# B&R Automation Studio project EFI (part 21)

#### AlarmsSummary.st
```iecst
ACTION AlarmsSummary:

	gMachine.Al.xAlrDisableGoToProduction := FALSE;

	IF gMachine.Pt.CT.iNumBlocks = 1 THEN
		gMachine.Al.xAlrSafetySystemEStop:=	gBlock[1].Al.xAlrEmergencyStop;
	ELSIF gMachine.Pt.CT.iNumBlocks = 2 THEN
		gMachine.Al.xAlrSafetySystemEStop:= gBlock[1].Al.xAlrEmergencyStop OR gBlock[2].Al.xAlrEmergencyStop;
	END_IF

	iReasonSafetySystemGeneral.0 := gMachine.Al.xAlrSafetySystemEStop;
	iReasonSafetySystemGeneral.1 := gBlock[1].AlSummary.xAlrSafetySystemGeneral AND gBlock[1].parSw.xEnableToMovements;
	iReasonSafetySystemGeneral.2 := gBlock[2].AlSummary.xAlrSafetySystemGeneral AND gBlock[2].parSw.xEnableToMovements;
	iReasonSafetySystemGeneral.3 := gMachine.Al.Alarm.xAlrSafetyNotEnabled;
	gMachine.AlSummary.xAlrSafetySystemGeneral:= iReasonSafetySystemGeneral > 0;

	iReasonSafetyCutAir.0 := gBlock[1].AlSummary.xAlrSafetyCutAir AND gBlock[1].parSw.xEnableToMovements;
	iReasonSafetyCutAir.1 := gBlock[2].AlSummary.xAlrSafetyCutAir AND gBlock[2].parSw.xEnableToMovements;
	gMachine.AlSummary.xAlrSafetyCutAir:= iReasonSafetyCutAir > 0;

	//////////////////
	// General Summary
	//////////////////

	//Silvia: any general warning+any block warning+any inks warning+any photocell warning.
	//Warnings//
	reasonAnyWarningGen.0 := gMachine.Al.Warning.xNotLoadedImage;
	reasonAnyWarningGen.1 := gMachine.Al.Alarm.xAlarmPlarformInc;
	reasonAnyWarningGen.2 := gMachine.Al.Alarm.xNoActionDangerCollision;
	reasonAnyWarningGen.3 := gMachine.Al.Warning.xBentTile;
	reasonAnyWarningGen.4 := gMachine.Al.Warning.xMaxMovsBentTile;
	reasonAnyWarningGen.5 := gMachine.Al.Alarm.xAlarmNotInPrintPosition;
	reasonAnyWarningGen.6 := gMachine.Al.Warning.xExternalCleanActive;
	reasonAnyWarningGen.7 := gMachine.Al.Warning.xSAIFault;
	reasonAnyWarningGen.8 := gMachine.Al.Warning.xSAIBypass;
	reasonAnyWarningGen.9 := gMachine.Al.Warning.xSAILowBat;
	reasonAnyWarningGen.10 := gMachine.Al.Warning.xValidConfiguration;
	reasonAnyWarningGen.11 := gBelt.AlSummary.xAnyWarning;
	reasonAnyWarningGen.12 := gBlock[1].AlSummary.xAnyWarning;
	reasonAnyWarningGen.13 := gBlock[2].AlSummary.xAnyWarning;
	reasonAnyWarningGen.14 := gPhotoCells.AlSummary.xAnyWarning;
	reasonAnyWarningGen.15 := gMachine.Al.Warning.xPCCabineSensAlrm;
	reasonAnyWarningGen.16 := gCuringLed[iIndexWhiteCuringLedBar].AlSummary.xAnyWarning;
	reasonAnyWarningGen.17 := gCuringLed[iIndexColorCuringLedBar].AlSummary.xAnyWarning;
	reasonAnyWarningGen.18 := gTransVacuum[1].AlSummary.xAnyWarning;
	reasonAnyWarningGen.19 := gTransVacuum[2].AlSummary.xAnyWarning;
	reasonAnyWarningGen.20 := gMachine.parSw.UI.xWarningCondition;
	reasonAnyWarningGen.21 := gMachine.Al.Warning.xNoCleaningModeEnabled;
	reasonAnyWarningGen.22 := gMachine.Al.Warning.xMediaIncoherenceDetectedL1;
	reasonAnyWarningGen.23 := gMachine.Al.Warning.xMediaIncoherenceDetectedL2;
	reasonAnyWarningGen.24 := gMachine.Al.Warning.xAlrHoopersSoftStarterFault;
	reasonAnyWarningGen.25 := gMachine.Al.Warning.xOvervoltage;
	reasonAnyWarningGen.25 := gBeltClean.AlSummary.xAnyAlarm;
	reasonAnyWarningGen.26 := gMachine.Al.Warning.xIonAntiStatic;
	reasonAnyWarningGen.27 := gMachine.Al.Warning.xErrorAntiStatic;
	reasonAnyWarningGen.28 := gMachine.Al.Warning.xWasteInkTankMaxLevelReached;

	reasonAnyWarningInks.0 := gInks[1].AlSummary.xAnyWarning;
	reasonAnyWarningInks.1 := gInks[2].AlSummary.xAnyWarning;
	reasonAnyWarningInks.2 := gInks[3].AlSummary.xAnyWarning;
	reasonAnyWarningInks.3 := gInks[4].AlSummary.xAnyWarning;
	reasonAnyWarningInks.4 := gInks[5].AlSummary.xAnyWarning;
	reasonAnyWarningInks.5 := gInks[6].AlSummary.xAnyWarning;
	reasonAnyWarningInks.6 := gInks[7].AlSummary.xAnyWarning;
	reasonAnyWarningInks.7 := gInks[8].AlSummary.xAnyWarning;
	reasonAnyWarningInks.8 := gInks[9].AlSummary.xAnyWarning;
	reasonAnyWarningInks.9 := gInks[10].AlSummary.xAnyWarning;
	reasonAnyWarningInks.10 := gInks[11].AlSummary.xAnyWarning;
	reasonAnyWarningInks.11 := gInks[12].AlSummary.xAnyWarning;

	gMachine.AlSummary.xAnyWarning:= reasonAnyWarningGen>0 OR reasonAnyWarningInks>0;

	//Any ALarm//
	gMachine.AlSummary.xAnyAlarm:= 	gMachine.AlSummary.xAlarmCritical OR
									gMachine.AlSummary.xAlarmStop;

	//Critial alarms//
	iReasonCritical.0 := gMachine.AlSummary.xAlrSafetySystemGeneral;
	iReasonCritical.1 := gMachine.Al.Alarm.xAlarmSAIPowerOff;
	iReasonCritical.2 := gBelt.AlSummary.xAlarmCritical;
	iReasonCritical.3 := gBlock[1].AlSummary.xAlarmCritical;
	iReasonCritical.4 := gBlock[2].AlSummary.xAlarmCritical;
	iReasonCritical.5 := gMachine.Al.Alarm.xAlrWrongPhysConf;
	iReasonCritical.6 := gMachine.Al.Alarm.xNoPowered;

	gMachine.AlSummary.CurrentReasonCritical := iReasonCritical;

	gMachine.AlSummary.xAlarmCritical:=  iReasonCritical > 0;
	//Register the reason of the Critical Alarm
	IF gMachine.St.Mode.xAuto AND EDGEPOS(gMachine.AlSummary.xAlarmCritical) THEN
		gMachine.AlSummary.iReasonCritical := iReasonCritical;
		LogCriticalAlarm;
	ELSIF EDGEPOS(gMachine.St.Mode.xAuto AND NOT gMachine.AlSummary.xAlarmCritical) THEN
		gMachine.AlSummary.iReasonCritical := 0;
	END_IF

	//Alarms stop//
	//Inks
	iReasonStopInks.0 := gInks[1].AlSummary.xAlarmStop;
	iReasonStopInks.1 := gInks[2].AlSummary.xAlarmStop;
	iReasonStopInks.2 := gInks[3].AlSummary.xAlarmStop;
	iReasonStopInks.3 := gInks[4].AlSummary.xAlarmStop;
	iReasonStopInks.4 := gInks[5].AlSummary.xAlarmStop;
	iReasonStopInks.5 := gInks[6].AlSummary.xAlarmStop;
	iReasonStopInks.6 := gInks[7].AlSummary.xAlarmStop;
	iReasonStopInks.7 := gInks[8].AlSummary.xAlarmStop;
	iReasonStopInks.8 := gInks[9].AlSummary.xAlarmStop;
	iReasonStopInks.9 := gInks[10].AlSummary.xAlarmStop;
	iReasonStopInks.10 := gInks[11].AlSummary.xAlarmStop;
	iReasonStopInks.11 := gInks[12].AlSummary.xAlarmStop;

	//General 1
	iReasonStopGen.0 := gMachine.Al.Alarm.xAlarmAir1;
	iReasonStopGen.1 := gMachine.Al.Alarm.xAlarmComPcPLC;
	iReasonStopGen.2 := gMachine.Al.Alarm.xAlarmEnableWithoutBarsOn;
	iReasonStopGen.3 := gMachine.Al.Alarm.xAlarmMountedPiece;
	iReasonStopGen.4 := gMachine.Al.Alarm.xAlarmSAIPowerFault;
	iReasonStopGen.5 := gMachine.Al.xAlrSafetySystemEStop;
	iReasonStopGen.6 := gMachine.Al.Alarm.xAlrThicknSystemNotSelected;
	iReasonStopGen.7 := gBlock[1].AlSummary.xAlarmStop;
	iReasonStopGen.8 := gBlock[2].AlSummary.xAlarmStop;
	iReasonStopGen.9 := gBelt.AlSummary.xAlarmStop;
	iReasonStopGen.10 := gDing.AlSummary.xAlarmStop;
	iReasonStopGen.11 := gPhotoCells.AlSummary.xAlarmStop;
	iReasonStopGen.12 := gTransVacuum[1].AlSummary.xAlarmStop;
	iReasonStopGen.13 := gTransVacuum[2].AlSummary.xAlarmStop;
	iReasonStopGen.14 := gMachine.Al.Alarm.xPDBrokenSensorL1;
	iReasonStopGen.15 := gMachine.Al.Alarm.xPDBrokenSensorL2;
	iReasonStopGen.16 := gJamDetect[1].AlSummary.xAlarmStop;
	iReasonStopGen.17 := gJamDetect[2].AlSummary.xAlarmStop;
	iReasonStopGen.18 := gNonCrash[1].AlSummary.xAlarmStop;
	iReasonStopGen.19 := gNonCrash[2].AlSummary.xAlarmStop;
	iReasonStopGen.20 := gMachine.Al.Alarm.xAlr24Vdc;
	//When printer is controlled by line, we consider curing led lamps errors in LineCtrl to execute a ControlledStop, but when printer is running by its own, must stop inmediately
	iReasonStopGen.21 := (gCuringLed[iIndexWhiteCuringLedBar].AlSummary.xAlarmStop OR gCuringLed[iIndexWhiteCuringLedBar].AlSummary.xAlarmCritical) AND NOT gMachine.Pt.xControlledByLine;
	iReasonStopGen.22 := (gCuringLed[iIndexColorCuringLedBar].AlSummary.xAlarmStop OR gCuringLed[iIndexColorCuringLedBar].AlSummary.xAlarmCritical) AND NOT gMachine.Pt.xControlledByLine;
	iReasonStopGen.23 := gMachine.Al.Alarm.xAlrDingWrongPosition;
	iReasonStopGen.24 := gMachine.Al.Alarm.xSwCriticalCondition;
	iReasonStopGen.25 := gJamDetect[3].AlSummary.xAlarmStop;
	iReasonStopGen.26 := gMachine.Al.Alarm.xNotLoadedImage;
	iReasonStopGen.27 := gThicknessCtrl.AlSummary.xAlarmStop;
	iReasonStopGen.28 := gMachine.Al.Alarm.xAlrThickOutLimits;
	iReasonStopGen.29 := gMachine.Al.Alarm.xAlrLengthOutLimits;
	iReasonStopGen.30 := gMachine.Al.Alarm.xAlrWidthOutLimits;

	gMachine.AlSummary.CurrentReasonStop[0] := iReasonStopInks;
	gMachine.AlSummary.CurrentReasonStop[1] := iReasonStopGen;

	gMachine.AlSummary.xAlarmStop:= iReasonStopGen > 0 OR iReasonStopInks > 0;
	//Register the reason of the Alarm
	IF NOT gMachine.St.AutoMode.xStop AND EDGEPOS(gMachine.AlSummary.xAlarmStop) THEN
		gMachine.AlSummary.iReasonStop[0] := iReasonStopInks;
		gMachine.AlSummary.iReasonStop[1] := iReasonStopGen;
		LogStopAlarm;
	ELSIF EDGEPOS(NOT gMachine.St.AutoMode.xStop AND NOT gMachine.AlSummary.xAlarmStop) THEN
		gMachine.AlSummary.iReasonStop[0] := 0;
		gMachine.AlSummary.iReasonStop[1] := 0;
	END_IF

END_ACTION
```

#### MachineInputs.st
```iecst
ACTION MachineInputs:

	// Product Detect. Manage general signal from signal connected to any block

	//Aggregated signals in the machine to clarify reading code
	CASE gMachine.Pt.PDSignalTpe OF
		PDCFG_CARRIAGE:
			// Check proper data assigned
			IF gMachine.In.ProductDetect.pPDCarriageSignalL1 = 0 OR gMachine.In.ProductDetect.pPDCarriageSignalL2 = 0 THEN
				RETURN;
			END_IF
			// Data pointer assignation
			xPDCarriageL1 ACCESS gMachine.In.ProductDetect.pPDCarriageSignalL1;
			xPDCarriageL2 ACCESS gMachine.In.ProductDetect.pPDCarriageSignalL2;
			// Status assignation
			gMachine.St.ProductDetect.xProductDetectL1 := xPDCarriageL1;
			gMachine.St.ProductDetect.xProductDetectL2 := xPDCarriageL2;

		PDCFG_SENSOR_AND_CARRIAGE,
		PDCFG_SENSOR:
			// Check proper data assigned
			IF gMachine.In.ProductDetect.pPDSignalSensorL1 = 0 OR ((gMachine.In.ProductDetect.pPDSignalSensorL2 = 0) AND gMachine.Pt.Hw.xDoubleLineAllowed) THEN
				RETURN;
			END_IF

			// Data pointer assignation
			xPDSignalSensorL1 ACCESS gMachine.In.ProductDetect.pPDSignalSensorL1;
			IF gMachine.Pt.Hw.xDoubleLineAllowed THEN
				xPDSignalSensorL2 ACCESS gMachine.In.ProductDetect.pPDSignalSensorL2;
			END_IF

			IF gThicknessCtrl.parameters.Detection.ProductDetect.xLoadMedia THEN
				gMachine.St.ProductDetect.xProductDetectL1 := gThicknessCtrl.status.Detection.xFilteredProductDetectMediaL1 AND gMachine.St.Position.xInPrint AND gMachine.parSw.Electronics.xRobotReadyL1;
				gMachine.St.ProductDetect.xProductDetectL2 := gThicknessCtrl.status.Detection.xFilteredProductDetectMediaL2 AND gMachine.St.Position.xInPrint AND gMachine.parSw.Electronics.xRobotReadyL2;
			ELSE
				//Status assignation
				gMachine.St.ProductDetect.xProductDetectL1 := xPDSignalSensorL1 AND gMachine.St.Position.xInPrint AND gMachine.parSw.Electronics.xRobotReadyL1;
				gMachine.St.ProductDetect.xProductDetectL2 := xPDSignalSensorL2 AND gMachine.St.Position.xInPrint AND gMachine.parSw.Electronics.xRobotReadyL2;
			END_IF

	END_CASE

	gMachine.St.ProductDetect.xAnyProductDetect := gMachine.St.ProductDetect.xProductDetectL1 OR gMachine.St.ProductDetect.xProductDetectL2;
	gMachine.St.ProductDetect.xAnyProductDetectDtpStricted := gMachine.St.ProductDetect.xProductDetectL1 OR (gMachine.St.ProductDetect.xProductDetectL2 AND gMachine.parSw.Dtp.xDoubleLine);

	gMachine.St.xMediaDetected := gDing.In.xDingLow OR gPhotoCells.status.xLowPieceDetect;

	//Counting edges of Product Detect sensor
	IF EDGEPOS(gMachine.St.ProductDetect.xProductDetectL1) THEN
		diCountProductDetectEdgesL1 := diCountProductDetectEdgesL1 + 1;
	END_IF
	IF EDGEPOS(gMachine.St.ProductDetect.xProductDetectL2) THEN
		diCountProductDetectEdgesL2 := diCountProductDetectEdgesL2 + 1;
	END_IF

	//Just for testing. To simulate media in real machine while degbugging with no real media available
	IF (gSimMachine.Commands.Media.xContinuousMediaPresent AND gBelt.states.xRuningBelt) THEN
		xBeltSpeedChanged 	:= rPrevBeltSpeed <> gBelt.states.rCurrentSpeed;
		xFormatChanged 		:= 	rPrevBoardLength <> gMachine.parSw.Media.rLength OR
								rPrevBoardGap <> gMachine.parSw.Media.rGap;

		IF (xBeltSpeedChanged OR xFormatChanged) AND (gBelt.states.rCurrentSpeed > gc_rMinSpeedToStart) THEN
			rBeltSpeedMmMs := (gBelt.states.rCurrentSpeed/60);

			//Board
			tiBoardTime := REAL_TO_TIME(gMachine.parSw.Media.rLength/rBeltSpeedMmMs);
			tiGapTime := REAL_TO_TIME(gMachine.parSw.Media.rGap/rBeltSpeedMmMs);

		END_IF
		rPrevBeltSpeed := gBelt.states.rCurrentSpeed;
		rPrevBoardLength := gMachine.parSw.Media.rLength;
		rPrevBoardGap := gMachine.parSw.Media.rGap;
		rPrevStainLength := gSimMachine.Parameters.rStainLength;
		rPrevStainGap := gSimMachine.Parameters.rStainGap;

		//To simulate a media
		BoardsFeedMinGap.tTimeOn := tiBoardTime;
		BoardsFeedMinGap.tTimeOff := tiGapTime;
		BoardsFeedMinGap.xEnable := TRUE;
	ELSE
		BoardsFeedMinGap.xEnable := FALSE;
	END_IF
	BoardsFeedMinGap();
END_ACTION
```

#### ResetAlarms.st
```iecst
ACTION ResetAlarms:

	gMachine.Al:=stPrinterAlarmsReseted;
	gMachine.Al.Alarm:= stPrinterAlarmsListReseted;

END_ACTION
```

- MachineStates.graphml - YED documentation (not shown)

### Program Logical/Printer/PhysicalMapping/PhysicalMapInputs (IEC) - Inputs program

#### Variables.var
```iecst
VAR
	T_Mute : TOF;
	T_Reset : TON;
	iIndexBlock : USINT;
	iIndexVac : USINT;
	iIndexCuringLed : USINT;
END_VAR
```

#### InputsNozomi2.st
```iecst
ACTION InputsNozomi2:

	//////////
	//PRINTER
	//////////

	// Machine controlled by line. Always with consent
	gMachine.In.xConsentL1Ok := TRUE;
	gMachine.In.xConsentL2Ok := TRUE;

	//Digital Inputs
	gMachine.In.Buttons.xStart := X20DIF371_101.DInput[1];
	gMachine.In.Buttons.xStop := NOT X20DIF371_101.DInput[2];
	gMachine.In.Buttons.xAuto := X20DIF371_101.DInput[3];
	gMachine.In.Buttons.xZero := NOT X20DIF371_101.DInput[4];
	gMachine.In.Buttons.xManual := X20DIF371_101.DInput[5];
	gMachine.In.Buttons.xReset := X20DIF371_101.DInput[6];

	gMachine.In.ProductDetect.pPDCarriageSignalL1 := ADR(X20DIF371_101.DInput[7]);
	gMachine.In.ProductDetect.pPDCarriageSignalL2 := ADR(X20DIF371_101.DInput[8]);
	gMachine.In.ProductDetect.pPDCarriage2SignalL1 := ADR(X20DIF371_101.DInput[9]);
	gMachine.In.ProductDetect.pPDCarriage2SignalL2 := ADR(X20DIF371_101.DInput[10]);

	//Jam device N3
	gJamInputs[3].xJamLowCrash := X20DIF371_101.DInput[11];
	gJamInputs[3].xJamTestOk := X20DIF371_101.DInput[12];
	gJamInputs[3].xJamCrash[1] := X20DIF371_101.DInput[13];

	gInksInputs[1].xPrintHeadsPsuOK := X20DIF371_102.DInput[1];
	gInksInputs[2].xPrintHeadsPsuOK := X20DIF371_102.DInput[2];
	gInksInputs[3].xPrintHeadsPsuOK := X20DIF371_102.DInput[3];
	gInksInputs[4].xPrintHeadsPsuOK := X20DIF371_102.DInput[4];
	gInksInputs[5].xPrintHeadsPsuOK := X20DIF371_102.DInput[5];
	gInksInputs[6].xPrintHeadsPsuOK := X20DIF371_102.DInput[6];
	gInksInputs[7].xPrintHeadsPsuOK := X20DIF371_102.DInput[7];
	gInksInputs[8].xPrintHeadsPsuOK := X20DIF371_102.DInput[8];
	//SPARE := NOT X20DIF371_102.DInput[9];
	gBelt.parameters.xDriveProtectionOK := X20DIF371_102.DInput[10];
	gBlockInputs[1].xDriveProtectionOK := gBlockInputs[1].xDifferentialOK := X20DIF371_102.DInput[11];
	//Non-crash - CB contact alarm := X20DIF371_102.DInput[12];
	gMachine.In.x24Vdc := X20DIF371_102.DInput[13];
	gBlockInputs[1].xReferenceDI := X20DIF371_102.DInput[14];
	//Back Safety Key unlock - PRINTER := X20DIF371_102.DInput[15];
	gMachine.In.xCameraDefectDetected := X20DIF371_102.DInput[16];

	IF NOT gMachine.St.HwData.xUpsOutOfPrinter THEN
		gMachine.In.UPSs[1].LoadOnUtility	:= X20DIF371_103.DInput[1];
		gMachine.In.UPSs[1].LoadOnBattery 	:= gMachine.In.UPSs[1].xPowerFault := X20DIF371_103.DInput[2]; //To review why name of signal is different for S1400 than Nz2. Signal coming from ups has same behaviour
		gMachine.In.UPSs[1].xLowBattery 	:= X20DIF371_103.DInput[3];
		gMachine.In.UPSs[1].xByPass 		:= X20DIF371_103.DInput[4];
		gMachine.In.UPSs[2].LoadOnUtility	:= X20DIF371_103.DInput[5];
		gMachine.In.UPSs[2].LoadOnBattery 	:= gMachine.In.UPSs[2].xPowerFault := X20DIF371_103.DInput[6]; //To review why name of signal is different for S1400 than Nz2. Signal coming from ups has same behaviour
		gMachine.In.UPSs[2].xLowBattery 	:= X20DIF371_103.DInput[7];
		gMachine.In.UPSs[2].xByPass 		:= X20DIF371_103.DInput[8];
	END_IF

	gMachine.In.ProductDetect.pPDSignalSensorL1	:= ADR(X20DIF371_103.DInput[9]);
	gMachine.In.ProductDetect.pPDSignalSensorL2	:= ADR(X20DIF371_103.DInput[10]);
//	gPhotoCells.Inputs.Signals.xPhotoCells[1] := NOT X20DIF371_103.DInput[11]; //Signal moved to FastInputs program
//	gPhotoCells.Inputs.Signals.xPhotoCells[2] := NOT X20DIF371_103.DInput[12]; //Signal moved to FastInputs program
//	gPhotoCells.Inputs.Signals.xPhotoCells[3] := NOT X20DIF371_103.DInput[13]; //Signal moved to FastInputs program
//	gPhotoCells.Inputs.Signals.xPhotoCells[4] := NOT X20DIF371_103.DInput[14]; //Signal moved to FastInputs program
//	gPhotoCells.Inputs.Signals.xPhotoCells[5] := NOT X20DIF371_103.DInput[15]; //Signal moved to FastInputs program
//	gPhotoCells.Inputs.Signals.xPhotoCells[6] := NOT X20DIF371_103.DInput[16]; //Signal moved to FastInputs program

	gInksInputs[1].xKlixonTriggered := X20DIF371_104.DInput[1];
	gInksInputs[2].xKlixonTriggered := X20DIF371_104.DInput[2];
	gInksInputs[3].xKlixonTriggered := X20DIF371_104.DInput[3];
	gInksInputs[4].xKlixonTriggered := X20DIF371_104.DInput[4];
	gInksInputs[5].xKlixonTriggered := X20DIF371_104.DInput[5];
	gInksInputs[6].xKlixonTriggered := X20DIF371_104.DInput[6];
	gInksInputs[7].xKlixonTriggered := X20DIF371_104.DInput[7];
	gInksInputs[8].xKlixonTriggered := X20DIF371_104.DInput[8];
	gJamInputs[1].xJamCrash[1] := X20DIF371_104.DInput[9];
	gJamInputs[1].xJamCrash[2] := X20DIF371_104.DInput[10];
	gJamInputs[1].xJamCrash[3] := X20DIF371_104.DInput[11];
	gJamInputs[1].xJamCrash[4] := X20DIF371_104.DInput[12];
	gJamInputs[2].xJamCrash[1] := X20DIF371_104.DInput[13];
	gJamInputs[2].xJamCrash[2] := X20DIF371_104.DInput[14];
	gJamInputs[2].xJamCrash[3] := X20DIF371_104.DInput[15];
	gJamInputs[2].xJamCrash[4] := X20DIF371_104.DInput[16];

	gInksInputs[1].xOverpressure  := NOT X20DIF371_105.DInput[1];
	gInksInputs[2].xOverpressure  := NOT X20DIF371_105.DInput[2];
	gInksInputs[3].xOverpressure  := NOT X20DIF371_105.DInput[3];
	gInksInputs[4].xOverpressure  := NOT X20DIF371_105.DInput[4];
	gInksInputs[5].xOverpressure  := NOT X20DIF371_105.DInput[5];
	gInksInputs[6].xOverpressure  := NOT X20DIF371_105.DInput[6];
	gInksInputs[7].xOverpressure  := NOT X20DIF371_105.DInput[7];
	gInksInputs[8].xOverpressure  := NOT X20DIF371_105.DInput[8];
	//Spare := X20DIF371_105.DInput[9];
	//Spare := X20DIF371_105.DInput[10];
	gMachine.In.xDegasserPressure := X20DIF371_105.DInput[11];
	gJamInputs[1].xJamLowCrash := X20DIF371_105.DInput[12];
	gJamInputs[2].xJamLowCrash := X20DIF371_105.DInput[13];
	gJamInputs[1].xJamTestOk := X20DIF371_105.DInput[14];
	gJamInputs[2].xJamTestOk := X20DIF371_105.DInput[15];
	FOR iIndexCuringLed:=1 TO MAX_LAST_CURING_LED DO
		gCuringLed[iIndexCuringLed].Signals.Inputs.xFrontDoorClosed := X20DIF371_105.DInput[16];
	END_FOR
	gBlockInputs[1].xFrontDoorClosed := X20DIF371_105.DInput[16];

	gBlockInputs[1].xPrintHeadPSU[1] := X20DI9372_107.DInput[1];
	gBlockInputs[1].xPrintHeadPSU[2] := X20DI9372_107.DInput[2];
	gBlockInputs[1].xPrintHeadPSU[3] := X20DI9372_107.DInput[3];
	gBlockInputs[1].xPrintHeadPSU[4] := X20DI9372_107.DInput[4];
	gBlockInputs[1].xPrintHeadPSU[5] := X20DI9372_107.DInput[5];
	gBlockInputs[1].xPrintHeadPSU[6] := X20DI9372_107.DInput[6];
	gBlockInputs[1].xHeaterDcOkBusBar1 := X20DI9372_107.DInput[7];
	gBlockInputs[1].xHeaterDcOkBusBar2 := X20DI9372_107.DInput[8];
	gMachine.In.xWasteInkTankMaxLevelReached := X20DI9372_107.DInput[9];

	//Analog inputs
	gInksInputs[1].iVacuum1Raw := X20AI8321_111.AInput[1];
	gInksInputs[1].xVacuum1SensorError 	:= StatusAnalogInputBroken( X20AI8321_111.ModuleOk, X20AI8321_111.Status01, X20AI8321_111.Status02, 1);
	gInksInputs[1].iVacuum2Raw := X20AI8321_111.AInput[2];
	gInksInputs[1].xVacuum2SensorError 	:= StatusAnalogInputBroken( X20AI8321_111.ModuleOk, X20AI8321_111.Status01, X20AI8321_111.Status02, 2);
	gInksInputs[2].iVacuum1Raw := X20AI8321_111.AInput[3];
	gInksInputs[2].xVacuum1SensorError 	:= StatusAnalogInputBroken( X20AI8321_111.ModuleOk, X20AI8321_111.Status01, X20AI8321_111.Status02, 3);
	gInksInputs[2].iVacuum2Raw := X20AI8321_111.AInput[4];
	gInksInputs[2].xVacuum2SensorError 	:= StatusAnalogInputBroken( X20AI8321_111.ModuleOk, X20AI8321_111.Status01, X20AI8321_111.Status02, 4);
	gInksInputs[3].iVacuum1Raw := X20AI8321_111.AInput[5];
	gInksInputs[3].xVacuum1SensorError 	:= StatusAnalogInputBroken( X20AI8321_111.ModuleOk, X20AI8321_111.Status01, X20AI8321_111.Status02, 5);
	gInksInputs[3].iVacuum2Raw := X20AI8321_111.AInput[6];
	gInksInputs[3].xVacuum2SensorError 	:= StatusAnalogInputBroken( X20AI8321_111.ModuleOk, X20AI8321_111.Status01, X20AI8321_111.Status02, 6);
	gInksInputs[4].iVacuum1Raw := X20AI8321_111.AInput[7];
	gInksInputs[4].xVacuum1SensorError 	:= StatusAnalogInputBroken( X20AI8321_111.ModuleOk, X20AI8321_111.Status01, X20AI8321_111.Status02, 7);
	gInksInputs[4].iVacuum2Raw := X20AI8321_111.AInput[8];
	gInksInputs[4].xVacuum2SensorError 	:= StatusAnalogInputBroken( X20AI8321_111.ModuleOk, X20AI8321_111.Status01, X20AI8321_111.Status02, 8);

	gInksInputs[5].iVacuum1Raw := X20AI8321_112.AInput[1];
	gInksInputs[5].xVacuum1SensorError 	:= StatusAnalogInputBroken( X20AI8321_112.ModuleOk, X20AI8321_112.Status01, X20AI8321_112.Status02, 1);
	gInksInputs[5].iVacuum2Raw := X20AI8321_112.AInput[2];
	gInksInputs[5].xVacuum2SensorError 	:= StatusAnalogInputBroken( X20AI8321_112.ModuleOk, X20AI8321_112.Status01, X20AI8321_112.Status02, 2);
	gInksInputs[6].iVacuum1Raw := X20AI8321_112.AInput[3];
	gInksInputs[6].xVacuum1SensorError 	:= StatusAnalogInputBroken( X20AI8321_112.ModuleOk, X20AI8321_112.Status01, X20AI8321_112.Status02, 3);
	gInksInputs[6].iVacuum2Raw := X20AI8321_112.AInput[4];
	gInksInputs[6].xVacuum2SensorError 	:= StatusAnalogInputBroken( X20AI8321_112.ModuleOk, X20AI8321_112.Status01, X20AI8321_112.Status02, 4);
	gInksInputs[7].iVacuum1Raw := X20AI8321_112.AInput[5];
	gInksInputs[7].xVacuum1SensorError 	:= StatusAnalogInputBroken( X20AI8321_112.ModuleOk, X20AI8321_112.Status01, X20AI8321_112.Status02, 5);
	gInksInputs[7].iVacuum2Raw := X20AI8321_112.AInput[6];
	gInksInputs[7].xVacuum2SensorError 	:= StatusAnalogInputBroken( X20AI8321_112.ModuleOk, X20AI8321_112.Status01, X20AI8321_112.Status02, 6);
	gInksInputs[8].iVacuum1Raw := X20AI8321_112.AInput[7];
	gInksInputs[8].xVacuum1SensorError 	:= StatusAnalogInputBroken( X20AI8321_112.ModuleOk, X20AI8321_112.Status01, X20AI8321_112.Status02, 7);
	gInksInputs[8].iVacuum2Raw := X20AI8321_112.AInput[8];
	gInksInputs[8].xVacuum2SensorError 	:= StatusAnalogInputBroken( X20AI8321_112.ModuleOk, X20AI8321_112.Status01, X20AI8321_112.Status02, 8);

	gTransVacuum[1].Inputs.iPressureRaw := X20AI8321_113.AInput[1];
	gTransVacuum[1].Inputs.xPressureSensorError := StatusAnalogInputBroken( X20AI8321_113.ModuleOk, X20AI8321_113.Status01, X20AI8321_113.Status02, 1);
	gTransVacuum[2].Inputs.iPressureRaw := X20AI8321_113.AInput[2];
	gTransVacuum[2].Inputs.xPressureSensorError := StatusAnalogInputBroken( X20AI8321_113.ModuleOk, X20AI8321_113.Status01, X20AI8321_113.Status02, 2);

	gInksInputs[2].iInTankLevel := X20AI8321_113.AInput[3];
	gInksInputs[2].xInkLevelTankSensorError := StatusAnalogInputBroken( X20AI8321_113.ModuleOk, X20AI8321_113.Status01, X20AI8321_113.Status02, 3);
	gInksInputs[3].iInTankLevel := X20AI8321_113.AInput[4];
	gInksInputs[3].xInkLevelTankSensorError := StatusAnalogInputBroken( X20AI8321_113.ModuleOk, X20AI8321_113.Status01, X20AI8321_113.Status02, 4);
	gInksInputs[4].iInTankLevel := X20AI8321_113.AInput[5];
	gInksInputs[4].xInkLevelTankSensorError := StatusAnalogInputBroken( X20AI8321_113.ModuleOk, X20AI8321_113.Status01, X20AI8321_113.Status02, 5);
	gInksInputs[5].iInTankLevel := X20AI8321_113.AInput[6];
	gInksInputs[5].xInkLevelTankSensorError := StatusAnalogInputBroken( X20AI8321_113.ModuleOk, X20AI8321_113.Status01, X20AI8321_113.Status02, 6);
	gInksInputs[6].iInTankLevel := X20AI8321_113.AInput[7];
	gInksInputs[6].xInkLevelTankSensorError := StatusAnalogInputBroken( X20AI8321_113.ModuleOk, X20AI8321_113.Status01, X20AI8321_113.Status02, 7);
	IF (gMachine.Pt.MachineModel = Type_NOZ_2_AQ) THEN
		gInksInputs[7].iInTankLevel := X20AI8321_113.AInput[8];
		gInksInputs[7].xInkLevelTankSensorError := StatusAnalogInputBroken( X20AI8321_113.ModuleOk, X20AI8321_113.Status01, X20AI8321_113.Status02, 8);
	ELSE
		gInksInputs[8].iInTankLevel := X20AI8321_113.AInput[8];
		gInksInputs[8].xInkLevelTankSensorError := StatusAnalogInputBroken( X20AI8321_113.ModuleOk, X20AI8321_113.Status01, X20AI8321_113.Status02, 8);
	END_IF

	//PT100
	gBlockInputs[1].xModuleTemp01Ok	:= X20AT4222_118.ModuleOk;
	gInksInputs[1].iTemperatureRaw := X20AT4222_118.TempInput[1];
	gInksInputs[1].xTempSensorError	:= StatusTemperatureInput(X20AT4222_118.Status01, 1);
	gInksInputs[2].iTemperatureRaw := X20AT4222_118.TempInput[2];
	gInksInputs[2].xTempSensorError	:= StatusTemperatureInput(X20AT4222_118.Status01, 2);
	gInksInputs[3].iTemperatureRaw := X20AT4222_118.TempInput[3];
	gInksInputs[3].xTempSensorError	:= StatusTemperatureInput(X20AT4222_118.Status01, 3);
	gInksInputs[4].iTemperatureRaw := X20AT4222_118.TempInput[4];
	gInksInputs[4].xTempSensorError	:= StatusTemperatureInput(X20AT4222_118.Status01, 4);

	gBlockInputs[1].xModuleTemp02Ok	:= X20AT4222_119.ModuleOk;
	gInksInputs[5].iTemperatureRaw := X20AT4222_119.TempInput[1];
	gInksInputs[5].xTempSensorError	:= StatusTemperatureInput(X20AT4222_119.Status01, 1);
	gInksInputs[6].iTemperatureRaw := X20AT4222_119.TempInput[2];
	gInksInputs[6].xTempSensorError	:= StatusTemperatureInput(X20AT4222_119.Status01, 2);
	gInksInputs[7].iTemperatureRaw := X20AT4222_119.TempInput[3];
	gInksInputs[7].xTempSensorError	:= StatusTemperatureInput(X20AT4222_119.Status01, 3);
	gInksInputs[8].iTemperatureRaw := X20AT4222_119.TempInput[4];
	gInksInputs[8].xTempSensorError	:= StatusTemperatureInput(X20AT4222_119.Status01, 4);

	// SI UNIT BK1
	gBlockInputs[1].xSiUnitModuleOk		:= SiUnitPwrLnkBK1.ModuleOk;
	gMachine.In.xAirSupply				:= SiUnitPwrLnkBK1.Input01_16.0;
	gBlockInputs[1].xAirVenturiOK		:= SiUnitPwrLnkBK1.Input01_16.1;
	gBlockInputs[1].xTrayOut			:= SiUnitPwrLnkBK1.Input01_16.2;
	gBlockInputs[1].xIclaSensor			:= SiUnitPwrLnkBK1.Input01_16.3;
	gTransVacuum[1].Inputs.xVaccAirFlow	:= gTransVacuum[2].Inputs.xVaccAirFlow := SiUnitPwrLnkBK1.Input01_16.4;
	gTransVacuum[1].Inputs.xJointSystemPressure:= gTransVacuum[2].Inputs.xJointSystemPressure := SiUnitPwrLnkBK1.Input01_16.5;
	gMachine.In.CleanBelt.xLowPosition 	:= SiUnitPwrLnkBK1.Input01_16.6;
	gMachine.In.CleanBelt.xHighPosition := SiUnitPwrLnkBK1.Input01_16.7;
	gBlockInputs[1].xBarsIn := TRUE;
	gTransVacuum[1].Inputs.xSafetyEnable := gTransVacuum[2].Inputs.xSafetyEnable := gMachine.In.xSafetyEnabled;

	//Signals Forced by Configuration
	gBlockInputs[1].Safety.xFrontEStopOK := gSafetyController.Inputs.xPrinterFrontsideEstop;
	gBlockInputs[1].Safety.xRearEStopOK := gSafetyController.Inputs.xPrinterBacksideEstop;

	gBlockInputs[1].Safety.xFrontSafetyOK	:= gSafetyController.Inputs.xPrinterFrontsideEstop AND gSafetyController.Inputs.xPrinterLightCurtain;
	gBlockInputs[1].Safety.xRearSafetyOK	:= gSafetyController.Inputs.xPrinterBacksideEstop AND gSafetyController.Inputs.xPrinterDoorLock;
	gBlockInputs[1].Safety.xSafetyOK 		:= gMachine.In.xSafetyEnabled;

	//There are no specific enables for light curtains. So we mapp PrinterLightCurtain status to these inputs to acknowledge that curtain is crossed
	gBlockInputs[1].Safety.xCurtainEnable01 := gBlockInputs[1].Safety.xCurtainEnable02 := gSafetyController.Inputs.xPrinterLightCurtain;

	//Signals Forced by Configuration
	FOR iIndexVac := 1 TO MAX_LAST_TRANS_VACUUM DO gTransVacuum[iIndexVac].Inputs.xBlowersAnyCB := FALSE; END_FOR

	///////////////////////////
	//UV Curing leds related

	//Digital inputs
	gCuringLed[iIndexColorCuringLedBar].Lamp[1].Inputs.ThermalFault	:= NOT X20DIF371_153.DInput[1];
	gCuringLed[iIndexColorCuringLedBar].Lamp[1].Inputs.SLMFault		:= NOT X20DIF371_153.DInput[2];
	gCuringLed[iIndexColorCuringLedBar].Lamp[2].Inputs.ThermalFault	:= NOT X20DIF371_153.DInput[3];
	gCuringLed[iIndexColorCuringLedBar].Lamp[2].Inputs.SLMFault		:= NOT X20DIF371_153.DInput[4];
	gCuringLed[iIndexColorCuringLedBar].Lamp[3].Inputs.ThermalFault	:= NOT X20DIF371_153.DInput[5];
	gCuringLed[iIndexColorCuringLedBar].Lamp[3].Inputs.SLMFault		:= NOT X20DIF371_153.DInput[6];
	gCuringLed[iIndexColorCuringLedBar].Lamp[4].Inputs.ThermalFault	:= NOT X20DIF371_153.DInput[7];
	gCuringLed[iIndexColorCuringLedBar].Lamp[4].Inputs.SLMFault		:= NOT X20DIF371_153.DInput[8];
	gCuringLed[iIndexColorCuringLedBar].Signals.Inputs.xN2HighFlow	:= NOT X20DIF371_153.DInput[9];
	gCuringLed[iIndexColorCuringLedBar].Signals.Inputs.xN2LowFlow		:= NOT X20DIF371_153.DInput[10];
	gMachine.In.AntiStatic.xGenAlarm								:= X20DIF371_153.DInput[13];
	gMachine.In.AntiStatic.xIonLevelAlarm							:= X20DIF371_153.DInput[14];

	gCuringLed[iIndexWhiteCuringLedBar].Lamp[1].Inputs.ThermalFault	:= NOT X20DIF371_154.DInput[1];
	gCuringLed[iIndexWhiteCuringLedBar].Lamp[1].Inputs.SLMFault		:= NOT X20DIF371_154.DInput[2];
	gCuringLed[iIndexWhiteCuringLedBar].Lamp[2].Inputs.ThermalFault	:= NOT X20DIF371_154.DInput[3];
	gCuringLed[iIndexWhiteCuringLedBar].Lamp[2].Inputs.SLMFault		:= NOT X20DIF371_154.DInput[4];
	gCuringLed[iIndexWhiteCuringLedBar].Lamp[3].Inputs.ThermalFault	:= NOT X20DIF371_154.DInput[5];
	gCuringLed[iIndexWhiteCuringLedBar].Lamp[3].Inputs.SLMFault		:= NOT X20DIF371_154.DInput[6];
	gCuringLed[iIndexWhiteCuringLedBar].Lamp[4].Inputs.ThermalFault	:= NOT X20DIF371_154.DInput[7];
	gCuringLed[iIndexWhiteCuringLedBar].Lamp[4].Inputs.SLMFault		:= NOT X20DIF371_154.DInput[8];
	gCuringLed[iIndexWhiteCuringLedBar].Signals.Inputs.xN2HighFlow	:= NOT X20DIF371_154.DInput[9];
	gCuringLed[iIndexWhiteCuringLedBar].Signals.Inputs.xN2LowFlow		:= NOT X20DIF371_154.DInput[10];

	gMachine.In.CleanBelt.xError := X20DIF371_154.DInput[13];

	gMachine.In.CleanBelt.xOpenGuide := X20DIF371_154.DInput[15]; //Clean Belt - Open Guide

	//Analog inputs
	gCuringLed[iIndexColorCuringLedBar].Lamp[1].Inputs.TemperatureRaw := X20AI8221_156.AInput[1];
	gCuringLed[iIndexColorCuringLedBar].Lamp[2].Inputs.TemperatureRaw := X20AI8221_156.AInput[2];
	gCuringLed[iIndexColorCuringLedBar].Lamp[3].Inputs.TemperatureRaw := X20AI8221_156.AInput[3];
	gCuringLed[iIndexColorCuringLedBar].Lamp[4].Inputs.TemperatureRaw := X20AI8221_156.AInput[4];
	gCuringLed[iIndexWhiteCuringLedBar].Lamp[1].Inputs.TemperatureRaw := X20AI8221_156.AInput[5];
	gCuringLed[iIndexWhiteCuringLedBar].Lamp[2].Inputs.TemperatureRaw := X20AI8221_156.AInput[6];
	gCuringLed[iIndexWhiteCuringLedBar].Lamp[3].Inputs.TemperatureRaw := X20AI8221_156.AInput[7];
	gCuringLed[iIndexWhiteCuringLedBar].Lamp[4].Inputs.TemperatureRaw := X20AI8221_156.AInput[8];

	//Edge hold down
	//Inductive sensors
	gPairedMotors[1].Motor[1].Inputs.xMinPositionReached := X20DIF371_180.DInput[1]; //Elevation motor. Entry side
	gPairedMotors[1].Motor[1].Inputs.xMaxPositionReached := X20DIF371_180.DInput[2]; //Elevation motor. Entry side
	gPairedMotors[2].Motor[1].Inputs.xMaxPositionReached := X20DIF371_180.DInput[3]; //Width fitting motor. Entry side
	gPairedMotors[2].Motor[1].Inputs.xMinPositionReached := X20DIF371_180.DInput[4]; //Width fitting motor. Entry side
	gPairedMotors[1].Motor[2].Inputs.xMinPositionReached := X20DIF371_180.DInput[5]; //Elevation motor. Exit side
	gPairedMotors[1].Motor[2].Inputs.xMaxPositionReached := X20DIF371_180.DInput[6]; //Elevation motor. Exit side
	gPairedMotors[2].Motor[2].Inputs.xMaxPositionReached := X20DIF371_180.DInput[7]; //Width fitting motor. Exit side
	gPairedMotors[2].Motor[2].Inputs.xMinPositionReached := X20DIF371_180.DInput[8]; //Width fitting motor. Exit side
	gEdgeHoldDown.inputs.xJam := NOT X20DIF371_180.DInput[9];
	gPairedMotors[1].Inputs.xSafetyEnable := gPairedMotors[2].Inputs.xSafetyEnable := gMachine.In.xSafetyEnabled;

	//Analog sensors
	gPairedMotors[2].Motor[1].Inputs.iMeasuredPositionFrontSide := X20AI8321_181.AInput[1];
	gPairedMotors[2].Motor[1].Inputs.xMeasuredPositionFrontSideError := StatusAnalogInputBroken( X20AI8321_181.ModuleOk, X20AI8321_181.Status01, X20AI8321_181.Status02, 1);
	gPairedMotors[2].Motor[1].Inputs.iMeasuredPositionBackSide := X20AI8321_181.AInput[2];
	gPairedMotors[2].Motor[1].Inputs.xMeasuredPositionBackSideError := StatusAnalogInputBroken( X20AI8321_181.ModuleOk, X20AI8321_181.Status01, X20AI8321_181.Status02, 2);
	gPairedMotors[2].Motor[2].Inputs.iMeasuredPositionFrontSide := X20AI8321_181.AInput[3];
	gPairedMotors[2].Motor[2].Inputs.xMeasuredPositionFrontSideError := StatusAnalogInputBroken( X20AI8321_181.ModuleOk, X20AI8321_181.Status01, X20AI8321_181.Status02, 3);
	gPairedMotors[2].Motor[2].Inputs.iMeasuredPositionBackSide := X20AI8321_181.AInput[4];
	gPairedMotors[2].Motor[2].Inputs.xMeasuredPositionBackSideError := StatusAnalogInputBroken( X20AI8321_181.ModuleOk, X20AI8321_181.Status01, X20AI8321_181.Status02, 4);

	//////////
	//PDC
	//////////
	//Line X20DIF371_002
	//These inputs are read in MachineConfigurator>InputsMachineModel
	//	:= Pdc_X20DIF371_002.DInput[1];
	//	:= Pdc_X20DIF371_002.DInput[2];
	//	:= Pdc_X20DIF371_002.DInput[3];
	//	:= Pdc_X20DIF371_002.DInput[4];
	//	:= Pdc_X20DIF371_002.DInput[5];
	//	:= Pdc_X20DIF371_002.DInput[6];
	gFeeder.Inputs.xNoPowered 					:= NOT Pdc_X20DIF371_002.DInput[7];
	gPrimer.Inputs.xNoPowered 					:= NOT Pdc_X20DIF371_002.DInput[8];
	gOverVarnish.Inputs.xNoPowered  			:= NOT Pdc_X20DIF371_002.DInput[9];
	gAxisInverter[1].ElecSignals.In.xBreakerOK 	:= Pdc_X20DIF371_002.DInput[10];
	gAxisInverter[2].ElecSignals.In.xBreakerOK 	:= Pdc_X20DIF371_002.DInput[11];
	gAxisInverter[3].ElecSignals.In.xBreakerOK 	:= Pdc_X20DIF371_002.DInput[12];
	gAxisInverter[4].ElecSignals.In.xBreakerOK 	:= Pdc_X20DIF371_002.DInput[13];
	gLine.Inputs.xPrinterPowered				:= Pdc_X20DIF371_002.DInput[14];
	gStacker.Inputs.xNoPowered 					:= NOT Pdc_X20DIF371_002.DInput[15];
	gLine.Inputs.xOvervoltageProtectionOk 		:= NOT Pdc_X20DIF371_002.DInput[16];

	//Line X20DIF371_003
	gMachine.In.xHoppersSoftStarterFault	:= Pdc_X20DIF371_003.DInput[1];
	gLine.Inputs.x24VdcStartSeqNoPowered	:= NOT Pdc_X20DIF371_003.DInput[2];
	gLine.Inputs.UPSs[1].LoadOnUtility		:= Pdc_X20DIF371_003.DInput[3];
	gLine.Inputs.UPSs[1].LoadOnBattery 		:= gLine.Inputs.UPSs[1].xPowerFault := Pdc_X20DIF371_003.DInput[4];
	gLine.Inputs.UPSs[1].xLowBattery 		:= Pdc_X20DIF371_003.DInput[5];
	gLine.Inputs.UPSs[1].xByPass			:= Pdc_X20DIF371_003.DInput[6];
	//Maneta printer accionada				:= Pdc_X20DIF371_003.DInput[7];		**To be check with HW team
	gChiller[1].In.xCooling					:= Pdc_X20DIF371_003.DInput[8]; // NOZOMITWO-1410
	gChiller[1].In.xPowered					:= Pdc_X20DIF371_003.DInput[9]; // NOZOMITWO-1410
	gChiller[1].In.xAlarm					:= NOT Pdc_X20DIF371_003.DInput[10]; // NOZOMITWO-1410
	//SPARE := Pdc_X20DIF371_003.DInput[11];
	//SPARE := Pdc_X20DIF371_003.DInput[12];
	//SPARE := Pdc_X20DIF371_003.DInput[13];
	//SPARE := Pdc_X20DIF371_003.DInput[14];

	//Line X20DIF371_004
	//Main Switch Accionado - Dryer 	:= Pdc_X20DIF371_004.DInput[1];	**To be check with HW team
	gDryerAnc.Inputs.xError 			:= Pdc_X20DIF371_004.DInput[2];
	gFeeder.Inputs.xOnline 				:= Pdc_X20DIF371_004.DInput[3];
	gFeeder.Inputs.xError 				:= Pdc_X20DIF371_004.DInput[4];
	gFeeder.Inputs.xFeeding 			:= Pdc_X20DIF371_004.DInput[5];
	gFeeder.Inputs.xMultiPick 			:= Pdc_X20DIF371_004.DInput[6];
	gFeeder.Inputs.xTrayEmpty 			:= Pdc_X20DIF371_004.DInput[7];
	gFeeder.Inputs.xMediaLowL1 			:= Pdc_X20DIF371_004.DInput[8];
	gFeeder.Inputs.xMediaThickness 		:= Pdc_X20DIF371_004.DInput[9];
	gFeeder.Inputs.xReadyToFeed 		:= Pdc_X20DIF371_004.DInput[10];
	gFeeder.Inputs.xModelInput[0] 		:= Pdc_X20DIF371_004.DInput[11];
	gFeeder.Inputs.xModelInput[1] 		:= Pdc_X20DIF371_004.DInput[12];
	gFeeder.Inputs.xModelInput[2] 		:= Pdc_X20DIF371_004.DInput[13];
	gPrimer.Inputs.xReadyToPrime 		:= Pdc_X20DIF371_004.DInput[14];
	gPrimer.Inputs.xCoating 			:= Pdc_X20DIF371_004.DInput[15];
	gPrimer.Inputs.xError 				:= Pdc_X20DIF371_004.DInput[16];

	//Line X20DIF371_005
	gPrimer.Inputs.xDryerInRun 			:= Pdc_X20DIF371_005.DInput[1];
	gPrimer.Inputs.xTransportMoving 	:= Pdc_X20DIF371_005.DInput[2];
	gPrimer.Inputs.xModelInput[0] 		:= Pdc_X20DIF371_005.DInput[3];
	gPrimer.Inputs.xModelInput[1] 		:= Pdc_X20DIF371_005.DInput[4];
	gPrimer.Inputs.xModelInput[2] 		:= Pdc_X20DIF371_005.DInput[5];
	gOverVarnish.Inputs.xReadyToPrime 	:= Pdc_X20DIF371_005.DInput[6];
	gOverVarnish.Inputs.xCoating 		:= Pdc_X20DIF371_005.DInput[7];
	gOverVarnish.Inputs.xError 			:= Pdc_X20DIF371_005.DInput[8];
	gOverVarnish.Inputs.xDryerInRun 	:= Pdc_X20DIF371_005.DInput[9];
	gOverVarnish.Inputs.xTransportMoving := Pdc_X20DIF371_005.DInput[10];
	gOverVarnish.Inputs.xModelInput[0] 	:= Pdc_X20DIF371_005.DInput[11];
	gOverVarnish.Inputs.xModelInput[1] 	:= Pdc_X20DIF371_005.DInput[12];
	gOverVarnish.Inputs.xModelInput[2] 	:= Pdc_X20DIF371_005.DInput[13];
	gDryerAnc.Inputs.xModelInput[0] 	:= Pdc_X20DIF371_005.DInput[14];
	gDryerAnc.Inputs.xModelInput[1] 	:= Pdc_X20DIF371_005.DInput[15];
	gDryerAnc.Inputs.xModelInput[2] 	:= Pdc_X20DIF371_005.DInput[16];

	//Line X20DIF371_006
	gStacker.Inputs.xError 				:= Pdc_X20DIF371_006.DInput[1];
	gStacker.Inputs.xReadyToStack 		:= Pdc_X20DIF371_006.DInput[2];
	gStacker.Inputs.xFeedInterrupt 		:= Pdc_X20DIF371_006.DInput[3];
	gStacker.Inputs.xRunning 			:= Pdc_X20DIF371_006.DInput[4];
	gStacker.Inputs.xModelInput[0] 		:= Pdc_X20DIF371_006.DInput[5];
	gStacker.Inputs.xModelInput[1] 		:= Pdc_X20DIF371_006.DInput[6];
	gStacker.Inputs.xModelInput[2] 		:= Pdc_X20DIF371_006.DInput[7];
	gStacker.Inputs.xRejectSuccess 		:= Pdc_X20DIF371_006.DInput[8];
	gStacker.Inputs.xStackSuccess 		:= Pdc_X20DIF371_006.DInput[9];

	gMachine.In.xRemoteJog 				:= Pdc_X20DIF371_006.DInput[11];

	//SPARE := Pdc_X20DIF371_006.DInput[10];
	//SPARE := Pdc_X20DIF371_006.DInput[11];
	//SPARE := Pdc_X20DIF371_006.DInput[12];
	//SPARE := Pdc_X20DIF371_006.DInput[13];
	//SPARE := Pdc_X20DIF371_006.DInput[14];
	gBeltClean.Inputs.xAirTurbVSDAvailable	:= Pdc_X20DIF371_006.DInput[15]; // NOZOMITWO-1912 New cleaning system for Noz2 water
	gMachine.In.xSafetyEnabled := Pdc_X20DIF371_006.DInput[16];

	//Line X20DIF371_020
	gCuringLed[iIndexColorCuringLedBar].Signals.Inputs.xPsuDcOk[1] := Pdc_X20DIF371_020.DInput[1];
	gCuringLed[iIndexColorCuringLedBar].Signals.Inputs.xPsuAcOk[1] := Pdc_X20DIF371_020.DInput[2];
	gCuringLed[iIndexColorCuringLedBar].Signals.Inputs.xPsuDcOk[2] := Pdc_X20DIF371_020.DInput[3];
	gCuringLed[iIndexColorCuringLedBar].Signals.Inputs.xPsuAcOk[2] := Pdc_X20DIF371_020.DInput[4];
	gCuringLed[iIndexColorCuringLedBar].Signals.Inputs.xPsuDcOk[3] := Pdc_X20DIF371_020.DInput[5];
	gCuringLed[iIndexColorCuringLedBar].Signals.Inputs.xPsuAcOk[3] := Pdc_X20DIF371_020.DInput[6];
	gCuringLed[iIndexColorCuringLedBar].Signals.Inputs.xPsuDcOk[4] := Pdc_X20DIF371_020.DInput[7];
	gCuringLed[iIndexColorCuringLedBar].Signals.Inputs.xPsuAcOk[4] := Pdc_X20DIF371_020.DInput[8];
	gCuringLed[iIndexColorCuringLedBar].Signals.Inputs.xPsuDcOk[5] := Pdc_X20DIF371_020.DInput[9];
	gCuringLed[iIndexColorCuringLedBar].Signals.Inputs.xPsuAcOk[5] := Pdc_X20DIF371_020.DInput[10];
	gCuringLed[iIndexColorCuringLedBar].Signals.Inputs.xPsuDcOk[6] := Pdc_X20DIF371_020.DInput[11];
	gCuringLed[iIndexColorCuringLedBar].Signals.Inputs.xPsuAcOk[6] := Pdc_X20DIF371_020.DInput[12];
	gCuringLed[iIndexColorCuringLedBar].Signals.Inputs.xSafetyEnable := gMachine.In.xSafetyEnabled;
	gChiller[gCuringLed[iIndexColorCuringLedBar].Parameters.iChillerIndex].In.xAlarm := Pdc_X20DIF371_020.DInput[16];

	//Line X20DIF371_021
	gCuringLed[iIndexWhiteCuringLedBar].Signals.Inputs.xPsuDcOk[1] := Pdc_X20DIF371_021.DInput[1];
	gCuringLed[iIndexWhiteCuringLedBar].Signals.Inputs.xPsuAcOk[1] := Pdc_X20DIF371_021.DInput[2];
	gCuringLed[iIndexWhiteCuringLedBar].Signals.Inputs.xPsuDcOk[2] := Pdc_X20DIF371_021.DInput[3];
	gCuringLed[iIndexWhiteCuringLedBar].Signals.Inputs.xPsuAcOk[2] := Pdc_X20DIF371_021.DInput[4];
	gCuringLed[iIndexWhiteCuringLedBar].Signals.Inputs.xPsuDcOk[3] := Pdc_X20DIF371_021.DInput[5];
	gCuringLed[iIndexWhiteCuringLedBar].Signals.Inputs.xPsuAcOk[3] := Pdc_X20DIF371_021.DInput[6];
	gCuringLed[iIndexWhiteCuringLedBar].Signals.Inputs.xPsuDcOk[4] := Pdc_X20DIF371_021.DInput[7];
	gCuringLed[iIndexWhiteCuringLedBar].Signals.Inputs.xPsuAcOk[4] := Pdc_X20DIF371_021.DInput[8];
	//Enable cleaning belt := Pdc_X20DIF371_021.DInput[9];
	gCuringLed[iIndexWhiteCuringLedBar].Signals.Inputs.xSafetyEnable := gMachine.In.xSafetyEnabled;
	gChiller[gCuringLed[iIndexWhiteCuringLedBar].Parameters.iChillerIndex].In.xAlarm := Pdc_X20DIF371_021.DInput[16];

	//Line X20DIF371_040
	gLine.Inputs.UPSs[2].LoadOnUtility			:= Pdc_X20DIF371_040.DInput[3];
	gLine.Inputs.UPSs[2].LoadOnBattery 			:= gLine.Inputs.UPSs[2].xPowerFault := Pdc_X20DIF371_040.DInput[4];
	gLine.Inputs.UPSs[2].xLowBattery 			:= Pdc_X20DIF371_040.DInput[5];
	gLine.Inputs.UPSs[2].xByPass				:= Pdc_X20DIF371_040.DInput[6];

	//Line X20DIF371_050 (Sarm related)
	gSarm.Inputs.xModelInput[0] := Pdc_X20DIF371_050.DInput[1];
	gSarm.Inputs.xModelInput[1] := Pdc_X20DIF371_050.DInput[2];
	gSarm.Inputs.xModelInput[2] := Pdc_X20DIF371_050.DInput[3];
	gSarm.Inputs.xError := Pdc_X20DIF371_050.DInput[4];
	gSarm.Inputs.xRunning := Pdc_X20DIF371_050.DInput[5];
	// := Pdc_X20DIF371_050.DInput[6];
	// := Pdc_X20DIF371_050.DInput[7];
	// := Pdc_X20DIF371_050.DInput[8];
	// := Pdc_X20DIF371_050.DInput[9];
	// := Pdc_X20DIF371_050.DInput[10];
	// := Pdc_X20DIF371_050.DInput[11];
	// := Pdc_X20DIF371_050.DInput[12];
	gSarm.Inputs.xPowered		:= Pdc_X20DIF371_050.DInput[13];
	//Primer "xNoPowered" input must be wired to the same input used for other ancillaries.
	gPrimer.Inputs.xIrPowered 	:= Pdc_X20DIF371_050.DInput[14]; //Mapped in case we would want raise alarm related to this power branch.
	gPrimer.Inputs.xUvPowered 	:= Pdc_X20DIF371_050.DInput[15]; //Mapped in case we would want raise alarm related to this power branch.
	//OverVarnish "xNoPowered" input must be wired to the same input used for other ancillaries.
	//gOverVarnish.Inputs.xNoPowered := NOT Pdc_X20DIF371_050.DInput[16];

	//Signals Forced by Configuration
	FOR iIndexBlock := 1 TO gMachine.Pt.CT.iNumBlocks DO
		gBlock[iIndexBlock].parameters.Hw.iNumPrintheadsPSU := 6;
		gBlock[iIndexBlock].parameters.Hw.iNumHeaterPSU := 0;
	END_FOR

	//To review with electrical team how to get these signals from chiller
	gChiller[1].In.xPowered	:= TRUE;
	gChiller[2].In.xPowered	:= TRUE;

END_ACTION
```

#### InputsP4.st
```iecst
ACTION InputsP4:

(* CABINET 01 *)

    // X1 PLC
	gMachine.In.xConsentL1Ok:= X1.DInput[1];
	gMachine.In.xConsentL2Ok:= X1.DInput[2];

	gMachine.In.xExternalCleaningOrder := X1.DInput[3];

	//Reserve01.DInput[1]:=X1.DInput[4];
	//Reserve01.AInput[1]:= X1.AInput[1];
	//Reserve01.AInput[2]:= X1.AInput[2];

	// X2 PLC
	//Reserve01.DInput[1]:= X2.DInput[1];
	//Reserve01.DInput[1]:= X2.DInput[2];
	//Reserve01.DInput[1]:= X2.DInput[3];
	//Reserve01.DInput[1]:= X2.DInput[4];
	gBelt.parameters.xDriveProtectionOK:= X2.DInput[5];
	//Reserve01.DInput[1]:= X2.DInput[6];
	//Reserve01.DInput[1]:= X2.DInput[7];
	//Reserve01.DInput[1]:= X2.DInput[8];
	//Reserve01.DInput[1]:= X2.DInput[9];

	// X3 PLC assignation to Laser detection
	gDing.In.xDingLow:= X3.DInput[5] AND gDing.State.xDingInstalled;
	gDing.In.xDingHigh:= X3.DInput[6] AND gDing.State.xDingInstalled;
	gDing.In.xModuleOK := X20AI2636_005.ModuleOk;
	gDing.In.xDingChannelFault := X20AI2636_005.DInput[1];

	// X2 PLC assignation to Photocell detection // FAST DETECTION
	// Those variables are not mapped. Are fast and assigned with pointer
	//gPhotoCells.Inputs.Signals.xPhotoCells[1] := NOT X2.DInput[11];	//It comes when X2 fast input
	//gPhotoCells.Inputs.Signals.xPhotoCells[2] := NOT X2.DInput[12];	// TRUE is not detecting tile
	//gPhotoCells.Inputs.Signals.xPhotoCells[3] := NOT X2.DInput[13];

	// X20DIF371_001
	gBlockInputs[1].xWaterLevelSensor	:=FALSE;
	gBlockInputs[1].xWaterPresureSensor :=FALSE;
	gBlockInputs[2].xWaterLevelSensor	:=FALSE;
	gBlockInputs[2].xWaterPresureSensor :=FALSE;

	// X20DIF371_002
	gMachine.In.UPSs[1].xPowerFault 	:= NOT X20DIF371_002.DInput[1];
	gMachine.In.UPSs[1].xByPass 		:= NOT X20DIF371_002.DInput[2];
	gMachine.In.UPSs[1].xLowBattery 		:= NOT X20DIF371_002.DInput[3];
	gMachine.In.UPSs[1].xSystemFault 	:= NOT X20DIF371_002.DInput[4];
	gMachine.In.UPSs[2].xPowerFault		:= NOT X20DIF371_002.DInput[5];
	gMachine.In.UPSs[2].xByPass			:= NOT X20DIF371_002.DInput[6];
	gMachine.In.UPSs[2].xLowBattery			:= NOT X20DIF371_002.DInput[7];
	gMachine.In.UPSs[2].xSystemFault	:= NOT X20DIF371_002.DInput[8];
	//Reserve01.DInput[1]				:= X20DIF371_002.DInput[9];
	gMachine.In.xPC1Ok				:= X20DIF371_002.DInput[10];
	gMachine.In.xPC2Ok				:= X20DIF371_002.DInput[11];
	gMachine.In.Buttons.xStart				:= X20DIF371_002.DInput[12];
	gMachine.In.Buttons.xStop				:= NOT X20DIF371_002.DInput[13];
	gMachine.In.Buttons.xAuto				:= X20DIF371_002.DInput[14];
	gMachine.In.Buttons.xManual				:= X20DIF371_002.DInput[15];
	//Reserve01.DInput[1]				:= X20DIF371_002.DInput[16];

	// X20DIF371_003										   (*scheme*)
	gMachine.In.Buttons.xZero:= NOT X20DIF371_003.DInput[1];	       (*DI0*)

	// gMachine.In.iMachineModelCode assigned in an specific Action

	//Reserve01.DInput[1]:= X20DIF371_003.DInput[8];
	//Reserve01.DInput[1]:= X20DIF371_003.DInput[9];
	//Reserve01.DInput[1]:= X20DIF371_003.DInput[10];
	//Reserve01.DInput[1]:= X20DIF371_003.DInput[11];
	//Reserve01.DInput[1]:= X20DIF371_003.DInput[12];
	//Reserve01.DInput[1]:= X20DIF371_003.DInput[13];
	//Reserve01.DInput[1]:= X20DIF371_003.DInput[14];
	//Reserve01.DInput[1]:= X20DIF371_003.DInput[15];
	gMachine.In.xTankHeaterPsuOK:= X20DIF371_003.DInput[16];

	// X20AI2636_005
	//NOTE: This code is in IN_Thickness program, to be sure to have it ready prior to work with it

	// Reset and Mute with the same digital signal
	T_Reset.IN := X20DIF371_002.DInput[16];
	T_Reset.PT := t#250ms;
	T_Reset();

	T_Mute.IN := X20DIF371_002.DInput[16];
	T_Mute.PT := t#100ms;
	T_Mute();

	gMachine.In.Buttons.xReset:= T_Reset.Q;
	gMachine.In.Buttons.xMute:= T_Mute.Q;

	// Transport enable with Released transport from Emegency Stops
	gMachine.In.xSafetyEnabled:= X20SLX402_006.DInput[10];

	// X20SM1436
	gPhotoCells.status.xBackModuleOk := X20SM1436_007.ModuleOk;
	gPhotoCells.status.xFrontModuleOk := X20SM1436_008.ModuleOk;

	// X20DIF371_030 pseudoSync/SYNC
	gMachine.In.xPbfCardOK := X20DIF371_030.ModuleOk;
	gMachine.In.iRelieve1.0:=X20DIF371_030.DInput[1];
	gMachine.In.iRelieve1.1:=X20DIF371_030.DInput[2];
	gMachine.In.iRelieve1.2:=X20DIF371_030.DInput[3];
	gMachine.In.iRelieve1.3:=X20DIF371_030.DInput[4];
	gMachine.In.iRelieve1.4:=X20DIF371_030.DInput[5];
	gMachine.In.iRelieve1.5:=X20DIF371_030.DInput[6];
	gMachine.In.iRelieve1.6:=X20DIF371_030.DInput[7];
	gMachine.In.iRelieve1.7:=X20DIF371_030.DInput[8];
	gMachine.In.iRelieve1.8:=X20DIF371_030.DInput[9];
	gMachine.In.iRelieve1.9 := FALSE;
	gMachine.In.iRelieve1.10:= FALSE;
	gMachine.In.iRelieve1.11:= FALSE;
	gMachine.In.iRelieve1.12:= FALSE;
	gMachine.In.iRelieve1.13:= FALSE;
	gMachine.In.iRelieve1.14:= FALSE;
	gMachine.In.iRelieve1.15:= FALSE;
	//Reserve01.DInput[1] := X20DIF371_030.DInput[10];
	//Reserve01.DInput[1] := X20DIF371_030.DInput[11];
	//Reserve01.DInput[1] := X20DIF371_030.DInput[12];
	//Reserve01.DInput[1] := X20DIF371_030.DInput[13];
	//Reserve01.DInput[1] := X20DIF371_030.DInput[14];
	//Reserve01.DInput[1] := X20DIF371_030.DInput[15];
	//Reserve01.DInput[1] := X20DIF371_030.DInput[16];

	// X20DIF371_101		(*  BAR A *) 	(*  BAR F *)
	gInksInputs[6].xMinLevel:= X20DIF371_101.DInput[1];
	gInksInputs[6].xMaxLevel:= X20DIF371_101.DInput[2];
	gInksInputs[5].xMinLevel:= X20DIF371_101.DInput[3];
	gInksInputs[5].xMaxLevel:= X20DIF371_101.DInput[4];
	gInksInputs[4].xMinLevel:= X20DIF371_101.DInput[5];
	gInksInputs[4].xMaxLevel:= X20DIF371_101.DInput[6];
	gInksInputs[3].xMinLevel:= X20DIF371_101.DInput[7];
	gInksInputs[3].xMaxLevel:= X20DIF371_101.DInput[8];
	gInksInputs[2].xMinLevel:= X20DIF371_101.DInput[9];
	gInksInputs[2].xMaxLevel:= X20DIF371_101.DInput[10];
	gInksInputs[1].xMinLevel:= X20DIF371_101.DInput[11];
	gInksInputs[1].xMaxLevel:= X20DIF371_101.DInput[12];
	gInksInputs[6].xOverpressure		:= NOT X20DIF371_101.DInput[13];
	gInksInputs[5].xOverpressure		:= NOT X20DIF371_101.DInput[14];
	gInksInputs[4].xOverpressure		:= NOT X20DIF371_101.DInput[15];
	gInksInputs[3].xOverpressure		:= NOT X20DIF371_101.DInput[16];

	// X20DIF371_102
	gInksInputs[2].xOverpressure		:= NOT X20DIF371_102.DInput[1];
	gInksInputs[1].xOverpressure		:= NOT X20DIF371_102.DInput[2];
	gBlockInputs[1].xDifferentialOK := X20DIF371_102.DInput[3];
	gBlockInputs[1].xDriveProtectionOK:= X20DIF371_102.DInput[4];
	gInksInputs[6].xPrintHeadsPsuOK		:= NOT X20DIF371_102.DInput[5];
	gInksInputs[5].xPrintHeadsPsuOK		:= NOT X20DIF371_102.DInput[6];
	gInksInputs[4].xPrintHeadsPsuOK		:= NOT X20DIF371_102.DInput[7];
	gInksInputs[3].xPrintHeadsPsuOK		:= NOT X20DIF371_102.DInput[8];
	gInksInputs[2].xPrintHeadsPsuOK		:= NOT X20DIF371_102.DInput[9];
	gInksInputs[1].xPrintHeadsPsuOK		:= NOT X20DIF371_102.DInput[10];
	gInksInputs[6].xKlixonTriggered  	:= X20DIF371_102.DInput[11];
	gInksInputs[5].xKlixonTriggered  	:= X20DIF371_102.DInput[12];
	gInksInputs[4].xKlixonTriggered  	:= X20DIF371_102.DInput[13];
	gInksInputs[3].xKlixonTriggered  	:= X20DIF371_102.DInput[14];
	gInksInputs[2].xKlixonTriggered  	:= X20DIF371_102.DInput[15];
	gInksInputs[1].xKlixonTriggered  	:= X20DIF371_102.DInput[16];

	// X20DIF371_103
	gBlockInputs[1].xWaterLevelSensor:= X20DIF371_103.DInput[1];
	gBlockInputs[1].xWaterPresureSensor:= X20DIF371_103.DInput[2];
	//Reserve01.DInput[1]:= X20DIF371_103.DInput[3];
	//Reserve01.DInput[1]:= X20DIF371_103.DInput[4];
	//Reserve01.DInput[1]:= X20DIF371_103.DInput[5];
	//Reserve01.DInput[1]:= X20DIF371_103.DInput[6];
	gBlockInputs[1].xHeaterDcOkBusBar1:= NOT X20DIF371_103.DInput[7];
	gBlockInputs[1].xReferenceDI:= X20DIF371_103.DInput[8];
	//Reserve01.DInput[1]:= X20DIF371_103.DInput[9];
	//Reserve01.DInput[1]:= X20DIF371_103.DInput[10];
	//Reserve01.DInput[1]:= X20DIF371_103.DInput[11];
	//Reserve01.DInput[1]:= X20DIF371_103.DInput[12];
	//Reserve01.DInput[1]:= X20DIF371_103.DInput[13];
	IF gBlock[1].parameters.iMappingBlock = 1 THEN
		gMachine.In.ProductDetect.pPDCarriageSignalL1 := ADR(X20DIF371_103.DInput[14]);
		gMachine.In.ProductDetect.pPDCarriageSignalL2 := ADR(X20DIF371_103.DInput[15]);
	END_IF
	//Reserve01.DInput[1]:= X20DIF371_103.DInput[16];

	// X20DC4395_104
	gInksInputs[6].iTachNegative		:= X20DC4395_104.CountInput[1];
	gInksInputs[4].iTachNegative		:= X20DC4395_104.CountInput[2];
	gInksInputs[2].iTachNegative		:= X20DC4395_104.CountInput[3];
	//Reserve01.DInput[1]:= X20DC4395_104.DInput[4];
	gInksInputs[5].iTachNegative		:= X20DC4395_104.CountInput[5];
	gInksInputs[3].iTachNegative		:= X20DC4395_104.CountInput[6];
	gInksInputs[1].iTachNegative		:= X20DC4395_104.CountInput[7];
	//Reserve01.DInput[1]:= X20DC4395_104.DInput[8];

	//  X20DC4395_105	(*  BAR A *) (*  BAR B *) (*  BAR C *) (*  BAR D *) (*  BAR E *) (*  BAR F *)
	gInksInputs[6].iTachFilling			:= X20DC4395_105.CountInput[1];
	gInksInputs[4].iTachFilling			:= X20DC4395_105.CountInput[2];
	gInksInputs[2].iTachFilling			:= X20DC4395_105.CountInput[3];
	//Reserve01.DInput[1]:= X20DC4395_105.DInput[4];
	gInksInputs[5].iTachFilling			:= X20DC4395_105.CountInput[5];
	gInksInputs[3].iTachFilling			:= X20DC4395_105.CountInput[6];
	gInksInputs[1].iTachFilling			:= X20DC4395_105.CountInput[7];
	//Reserve01.DInput[1]:= X20DC4395_105.DInput[8];

	// X20AI8321_109		(*  BAR A *) (*  BAR B *) (*  BAR C *) (*  BAR D *)
	gInksInputs[6].iVacuum1Raw			:= X20AI8321_109.AInput[1];
	gInksInputs[6].xVacuum1SensorError 	:= StatusAnalogInputBroken( X20AI8321_109.ModuleOk, X20AI8321_109.Status01, X20AI8321_109.Status02, 1);
	gInksInputs[6].iVacuum2Raw			:= X20AI8321_109.AInput[2];
	gInksInputs[6].xVacuum2SensorError 	:= StatusAnalogInputBroken( X20AI8321_109.ModuleOk, X20AI8321_109.Status01, X20AI8321_109.Status02, 2);
	gInksInputs[5].iVacuum1Raw			:= X20AI8321_109.AInput[3];
	gInksInputs[5].xVacuum1SensorError 	:= StatusAnalogInputBroken( X20AI8321_109.ModuleOk, X20AI8321_109.Status01, X20AI8321_109.Status02, 3);
	gInksInputs[5].iVacuum2Raw			:= X20AI8321_109.AInput[4];
	gInksInputs[5].xVacuum2SensorError 	:= StatusAnalogInputBroken( X20AI8321_109.ModuleOk, X20AI8321_109.Status01, X20AI8321_109.Status02, 4);
	gInksInputs[4].iVacuum1Raw			:= X20AI8321_109.AInput[5];
	gInksInputs[4].xVacuum1SensorError 	:= StatusAnalogInputBroken( X20AI8321_109.ModuleOk, X20AI8321_109.Status01, X20AI8321_109.Status02, 5);
	gInksInputs[4].iVacuum2Raw			:= X20AI8321_109.AInput[6];
	gInksInputs[4].xVacuum2SensorError 	:= StatusAnalogInputBroken( X20AI8321_109.ModuleOk, X20AI8321_109.Status01, X20AI8321_109.Status02, 6);
	gInksInputs[3].iVacuum1Raw			:= X20AI8321_109.AInput[7];
	gInksInputs[3].xVacuum1SensorError 	:= StatusAnalogInputBroken( X20AI8321_109.ModuleOk, X20AI8321_109.Status01, X20AI8321_109.Status02, 7);
	gInksInputs[3].iVacuum2Raw			:= X20AI8321_109.AInput[8];
	gInksInputs[3].xVacuum2SensorError 	:= StatusAnalogInputBroken( X20AI8321_109.ModuleOk, X20AI8321_109.Status01, X20AI8321_109.Status02, 8);

	// X20AI8321_110		(*  BAR E *) 	(*  BAR F *)
	gInksInputs[2].iVacuum1Raw			:= X20AI8321_110.AInput[1];
	gInksInputs[2].xVacuum1SensorError 	:= StatusAnalogInputBroken( X20AI8321_110.ModuleOk, X20AI8321_110.Status01, X20AI8321_110.Status02, 1);
	gInksInputs[2].iVacuum2Raw			:= X20AI8321_110.AInput[2];
	gInksInputs[2].xVacuum2SensorError 	:= StatusAnalogInputBroken( X20AI8321_110.ModuleOk, X20AI8321_110.Status01, X20AI8321_110.Status02, 2);
	gInksInputs[1].iVacuum1Raw			:= X20AI8321_110.AInput[3];
	gInksInputs[1].xVacuum1SensorError 	:= StatusAnalogInputBroken( X20AI8321_110.ModuleOk, X20AI8321_110.Status01, X20AI8321_110.Status02, 3);
	gInksInputs[1].iVacuum2Raw			:= X20AI8321_110.AInput[4];
	gInksInputs[1].xVacuum2SensorError 	:= StatusAnalogInputBroken( X20AI8321_110.ModuleOk, X20AI8321_110.Status01, X20AI8321_110.Status02, 4);
	//Reserve01.AInput[1]:= X20AI8321_110.AInput[5];
	//Reserve01.AInput[1]:= X20AI8321_110.AInput[6];
	//Reserve01.AInput[1]:= X20AI8321_110.AInput[7];
	//Reserve01.AInput[1]:= X20AI8321_110.AInput[8];

	// X20AT4222_114		(*  BAR A *) (*  BAR B *) (*  BAR C *) (*  BAR D *)  (*  BAR E *)  (*  BAR F *)

	gBlockInputs[1].xModuleTemp01Ok		:= X20AT4222_114.ModuleOk;
	gInksInputs[6].iTemperatureRaw  	:= X20AT4222_114.TempInput[1];
	gInksInputs[6].xTempSensorError		:= StatusTemperatureInput(X20AT4222_114.Status01, 1);
	gInksInputs[5].iTemperatureRaw  	:= X20AT4222_114.TempInput[2];
	gInksInputs[5].xTempSensorError		:= StatusTemperatureInput(X20AT4222_114.Status01, 2);
	gInksInputs[4].iTemperatureRaw  	:= X20AT4222_114.TempInput[3];
	gInksInputs[4].xTempSensorError		:= StatusTemperatureInput(X20AT4222_114.Status01, 3);
	gInksInputs[3].iTemperatureRaw  	:= X20AT4222_114.TempInput[4];
	gInksInputs[3].xTempSensorError		:= StatusTemperatureInput(X20AT4222_114.Status01, 4);

	// X20AT4222_115
	gBlockInputs[1].xModuleTemp02Ok			:= X20AT4222_115.ModuleOk;
	gInksInputs[2].iTemperatureRaw  		:= X20AT4222_115.TempInput[1];
	gInksInputs[2].xTempSensorError			:= StatusTemperatureInput(X20AT4222_115.Status01, 1);
	gInksInputs[1].iTemperatureRaw  		:= X20AT4222_115.TempInput[2];
	gInksInputs[1].xTempSensorError			:= StatusTemperatureInput(X20AT4222_115.Status01, 2);
	gInksInputs[6].iTemperatureTankRaw			:= X20AT4222_115.TempInput[3];
	gInksInputs[6].xTempTankSensorError	:= StatusTemperatureInput(X20AT4222_115.Status01, 3);
	gInksInputs[5].iTemperatureTankRaw			:= X20AT4222_115.TempInput[4];
	gInksInputs[5].xTempTankSensorError	:= StatusTemperatureInput(X20AT4222_115.Status01, 4);

	// X20AT4222_116
	gBlockInputs[1].xModuleTemp03Ok			:= X20AT4222_116.ModuleOk;
	gInksInputs[4].iTemperatureTankRaw			:= X20AT4222_116.TempInput[1];
	gInksInputs[4].xTempTankSensorError	:= StatusTemperatureInput(X20AT4222_116.Status01, 1);
	gInksInputs[3].iTemperatureTankRaw			:= X20AT4222_116.TempInput[2];
	gInksInputs[3].xTempTankSensorError	:= StatusTemperatureInput(X20AT4222_116.Status01, 2);
	gInksInputs[2].iTemperatureTankRaw			:= X20AT4222_116.TempInput[3];
	gInksInputs[2].xTempTankSensorError	:= StatusTemperatureInput(X20AT4222_116.Status01, 3);
	gInksInputs[1].iTemperatureTankRaw			:= X20AT4222_116.TempInput[4];
	gInksInputs[1].xTempTankSensorError	:= StatusTemperatureInput(X20AT4222_116.Status01, 4);

	// X20SI8110_117
	gBlockInputs[1].Safety.xRearEStopOK:=X20SI8110_117.DInput[1];
	gBlockInputs[1].Safety.xFrontEStopOK:=X20SI8110_117.DInput[3];
	gBlockInputs[1].Safety.xCurtainEnable01:=X20SI8110_117.DInput[5];
	gBlockInputs[1].Safety.xRearSafetyOK:=X20SI8110_117.DInput[6];
	gBlockInputs[1].Safety.xCurtainEnable02:=X20SI8110_117.DInput[7];

	// X20SO8110_118
	gBlockInputs[1].Safety.xSafetyOK:=X20SO2110_118.DInput[1];

	// SI UNIT BK1
	gBlockInputs[1].xSiUnitModuleOk:=SiUnitBK1.ModuleOk;  // Filter if it's necesary
	gMachine.In.xAirSupply:= SiUnitBK1.Input01_08.0;
	gBlockInputs[1].xAirVenturiOK:= SiUnitBK1.Input01_08.1;
	gBlockInputs[1].xTrayOut:= SiUnitBK1.Input01_08.2; // Out: Tray in safe position to move bars to print
	gBlockInputs[1].xIclaSensor:= SiUnitBK1.Input01_08.3;
	gBlockInputs[1].xBarsIn := TRUE;

	(* CABINET 03 *)

	// X20DIF371_201 		(*  BAR G *) 	(*  BAR L *)
	gInksInputs[12].xMinLevel:= X20DIF371_201.DInput[1];
	gInksInputs[12].xMaxLevel:= X20DIF371_201.DInput[2];
	gInksInputs[11].xMinLevel:= X20DIF371_201.DInput[3];
	gInksInputs[11].xMaxLevel:= X20DIF371_201.DInput[4];
	gInksInputs[10].xMinLevel:= X20DIF371_201.DInput[5];
	gInksInputs[10].xMaxLevel:= X20DIF371_201.DInput[6];
	gInksInputs[9].xMinLevel:=  X20DIF371_201.DInput[7];
	gInksInputs[9].xMaxLevel:=  X20DIF371_201.DInput[8];
	gInksInputs[8].xMinLevel:=  X20DIF371_201.DInput[9];
	gInksInputs[8].xMaxLevel:=  X20DIF371_201.DInput[10];
	gInksInputs[7].xMinLevel:=  X20DIF371_201.DInput[11];
	gInksInputs[7].xMaxLevel:=  X20DIF371_201.DInput[12];
	gInksInputs[12].xOverpressure := NOT X20DIF371_201.DInput[13];
	gInksInputs[11].xOverpressure := NOT X20DIF371_201.DInput[14];
	gInksInputs[10].xOverpressure := NOT X20DIF371_201.DInput[15];
	gInksInputs[9].xOverpressure  := NOT X20DIF371_201.DInput[16];

	// X20DIF371_202
	gInksInputs[8].xOverpressure := NOT X20DIF371_202.DInput[1];
	gInksInputs[7].xOverpressure := NOT X20DIF371_202.DInput[2];
	gBlockInputs[2].xDifferentialOK:= X20DIF371_202.DInput[3];
	gBlockInputs[2].xDriveProtectionOK:= X20DIF371_202.DInput[4];
	gInksInputs[12].xPrintHeadsPsuOK	:= NOT X20DIF371_202.DInput[5];
	gInksInputs[11].xPrintHeadsPsuOK	:= NOT X20DIF371_202.DInput[6];
	gInksInputs[10].xPrintHeadsPsuOK	:= NOT X20DIF371_202.DInput[7];
	gInksInputs[9].xPrintHeadsPsuOK		:= NOT X20DIF371_202.DInput[8];
	gInksInputs[8].xPrintHeadsPsuOK		:= NOT X20DIF371_202.DInput[9];
	gInksInputs[7].xPrintHeadsPsuOK		:= NOT X20DIF371_202.DInput[10];
	gInksInputs[12].xKlixonTriggered  	:= X20DIF371_202.DInput[11];
	gInksInputs[11].xKlixonTriggered  	:= X20DIF371_202.DInput[12];
	gInksInputs[10].xKlixonTriggered  	:= X20DIF371_202.DInput[13];
	gInksInputs[9].xKlixonTriggered  	:= X20DIF371_202.DInput[14];
	gInksInputs[8].xKlixonTriggered  	:= X20DIF371_202.DInput[15];
	gInksInputs[7].xKlixonTriggered  	:= X20DIF371_202.DInput[16];

	// X20DIF371_203
	//Reserve01.DInput[1]:= X20DIF371_203.DInput[1];
	//Reserve01.DInput[1]:= X20DIF371_203.DInput[2];
	//Reserve01.DInput[1]:= X20DIF371_203.DInput[3];
	//Reserve01.DInput[1]:= X20DIF371_203.DInput[4];
	//Reserve01.DInput[1]:= X20DIF371_203.DInput[5];
	//Reserve01.DInput[1]:= X20DIF371_203.DInput[6];
	gBlockInputs[2].xHeaterDcOkBusBar1:= NOT X20DIF371_203.DInput[7];
	gBlockInputs[2].xReferenceDI:= X20DIF371_203.DInput[8];
	//Reserve01.DInput[1]:= X20DIF371_203.DInput[9];
	//Reserve01.DInput[1]:= X20DIF371_203.DInput[10];
	//Reserve01.DInput[1]:= X20DIF371_203.DInput[11];
	//Reserve01.DInput[1]:= X20DIF371_203.DInput[12];
	//Reserve01.DInput[1]:= X20DIF371_203.DInput[13];
	IF gBlock[1].parameters.iMappingBlock = 2 THEN
		gMachine.In.ProductDetect.pPDCarriageSignalL1 := ADR(X20DIF371_203.DInput[14]);
		gMachine.In.ProductDetect.pPDCarriageSignalL2 := ADR(X20DIF371_203.DInput[15]);
	END_IF
	//Reserve01.DInput[1]:= X20DIF371_203.DInput[16];

	// X20DC4395_204
	gInksInputs[12].iTachNegative		:= X20DC4395_204.CountInput[1];
	gInksInputs[10].iTachNegative		:= X20DC4395_204.CountInput[2];
	gInksInputs[8].iTachNegative		:= X20DC4395_204.CountInput[3];
	//Reserve01.DInput[1]:= X20DC4395_204.DInput[4];
	gInksInputs[11].iTachNegative		:= X20DC4395_204.CountInput[5];
	gInksInputs[9].iTachNegative		:= X20DC4395_204.CountInput[6];
	gInksInputs[7].iTachNegative		:= X20DC4395_204.CountInput[7];
	//Reserve01.DInput[1]:= X20DC4395_204.DInput[8];

	//  X20DC4395_205	(*  BAR G *) (*  BAR H *) (*  BAR I *) (*  BAR J *) (*  BAR K *) (*  BAR L *)
	gInksInputs[12].iTachFilling		:= X20DC4395_205.CountInput[1];
	gInksInputs[10].iTachFilling		:= X20DC4395_205.CountInput[2];
	gInksInputs[8].iTachFilling			:= X20DC4395_205.CountInput[3];
	//Reserve01.DInput[1]:= X20DC4395_205.DInput[4];
	gInksInputs[11].iTachFilling		:= X20DC4395_205.CountInput[5];
	gInksInputs[9].iTachFilling			:= X20DC4395_205.CountInput[6];
	gInksInputs[7].iTachFilling			:= X20DC4395_205.CountInput[7];
	//Reserve01.DInput[1]:= X20DC4395_205.DInput[8];

	// X20AI8321_209	(*  BAR G *) (*  BAR H *) (*  BAR I *) (*  BAR J *)
	gInksInputs[12].iVacuum1Raw      	:= X20AI8321_209.AInput[1];
	gInksInputs[12].xVacuum1SensorError := StatusAnalogInputBroken( X20AI8321_209.ModuleOk, X20AI8321_209.Status01, X20AI8321_209.Status02, 1);
	gInksInputs[12].iVacuum2Raw      	:= X20AI8321_209.AInput[2];
	gInksInputs[12].xVacuum2SensorError := StatusAnalogInputBroken( X20AI8321_209.ModuleOk, X20AI8321_209.Status01, X20AI8321_209.Status02, 2);
	gInksInputs[11].iVacuum1Raw      	:= X20AI8321_209.AInput[3];
	gInksInputs[11].xVacuum1SensorError := StatusAnalogInputBroken( X20AI8321_209.ModuleOk, X20AI8321_209.Status01, X20AI8321_209.Status02, 3);
	gInksInputs[11].iVacuum2Raw      	:= X20AI8321_209.AInput[4];
	gInksInputs[11].xVacuum2SensorError := StatusAnalogInputBroken( X20AI8321_209.ModuleOk, X20AI8321_209.Status01, X20AI8321_209.Status02, 4);
	gInksInputs[10].iVacuum1Raw      	:= X20AI8321_209.AInput[5];
	gInksInputs[10].xVacuum1SensorError := StatusAnalogInputBroken( X20AI8321_209.ModuleOk, X20AI8321_209.Status01, X20AI8321_209.Status02, 5);
	gInksInputs[10].iVacuum2Raw      	:= X20AI8321_209.AInput[6];
	gInksInputs[10].xVacuum2SensorError := StatusAnalogInputBroken( X20AI8321_209.ModuleOk, X20AI8321_209.Status01, X20AI8321_209.Status02, 6);
	gInksInputs[9].iVacuum1Raw      	:= X20AI8321_209.AInput[7];
	gInksInputs[9].xVacuum1SensorError  := StatusAnalogInputBroken( X20AI8321_209.ModuleOk, X20AI8321_209.Status01, X20AI8321_209.Status02, 7);
	gInksInputs[9].iVacuum2Raw      	:= X20AI8321_209.AInput[8];
	gInksInputs[9].xVacuum2SensorError  := StatusAnalogInputBroken( X20AI8321_209.ModuleOk, X20AI8321_209.Status01, X20AI8321_209.Status02, 8);

	// X20AI8321_210 		(*  BAR K *)  (*  BAR L *)
	gInksInputs[8].iVacuum1Raw      	:= X20AI8321_210.AInput[1];
	gInksInputs[8].xVacuum1SensorError  := StatusAnalogInputBroken( X20AI8321_210.ModuleOk, X20AI8321_210.Status01, X20AI8321_210.Status02, 1);
	gInksInputs[8].iVacuum2Raw      	:= X20AI8321_210.AInput[2];
	gInksInputs[8].xVacuum2SensorError  := StatusAnalogInputBroken( X20AI8321_210.ModuleOk, X20AI8321_210.Status01, X20AI8321_210.Status02, 2);
	gInksInputs[7].iVacuum1Raw      	:= X20AI8321_210.AInput[3];
	gInksInputs[7].xVacuum1SensorError  := StatusAnalogInputBroken( X20AI8321_210.ModuleOk, X20AI8321_210.Status01, X20AI8321_210.Status02, 3);
	gInksInputs[7].iVacuum2Raw      	:= X20AI8321_210.AInput[4];
	gInksInputs[7].xVacuum2SensorError  := StatusAnalogInputBroken( X20AI8321_210.ModuleOk, X20AI8321_210.Status01, X20AI8321_210.Status02, 4);

	// X20AT4222_214		 (*  BAR G *)  (*  BAR H *)  (*  BAR I *)  (*  BAR J *)
	gBlockInputs[2].xModuleTemp01Ok		:= X20AT4222_214.ModuleOk;
	gInksInputs[12].iTemperatureRaw  	:= X20AT4222_214.TempInput[1];
	gInksInputs[12].xTempSensorError	:= StatusTemperatureInput(X20AT4222_214.Status01, 1);
	gInksInputs[11].iTemperatureRaw  	:= X20AT4222_214.TempInput[2];
	gInksInputs[11].xTempSensorError	:= StatusTemperatureInput(X20AT4222_214.Status01, 2);
	gInksInputs[10].iTemperatureRaw  	:= X20AT4222_214.TempInput[3];
	gInksInputs[10].xTempSensorError	:= StatusTemperatureInput(X20AT4222_214.Status01, 3);
	gInksInputs[9].iTemperatureRaw  	:= X20AT4222_214.TempInput[4];
	gInksInputs[9].xTempSensorError		:= StatusTemperatureInput(X20AT4222_214.Status01, 4);

	// X20AT4222_215 		(*  BAR K *)  (*  BAR L *)
	gBlockInputs[2].xModuleTemp02Ok			:= X20AT4222_215.ModuleOk;
	gInksInputs[8].iTemperatureRaw  		:= X20AT4222_215.TempInput[1];
	gInksInputs[8].xTempSensorError			:= StatusTemperatureInput(X20AT4222_215.Status01, 1);
	gInksInputs[7].iTemperatureRaw  		:= X20AT4222_215.TempInput[2];
	gInksInputs[7].xTempSensorError			:= StatusTemperatureInput(X20AT4222_215.Status01, 2);
	gInksInputs[12].iTemperatureTankRaw		:= X20AT4222_215.TempInput[3];
	gInksInputs[12].xTempTankSensorError	:= StatusTemperatureInput(X20AT4222_215.Status01, 3);
	gInksInputs[11].iTemperatureTankRaw		:= X20AT4222_215.TempInput[4];
	gInksInputs[11].xTempTankSensorError	:= StatusTemperatureInput(X20AT4222_215.Status01, 4);

	// X20AT4222_216
	gBlockInputs[2].xModuleTemp03Ok			:= X20AT4222_216.ModuleOk;
	gInksInputs[10].iTemperatureTankRaw		:= X20AT4222_216.TempInput[1];
	gInksInputs[10].xTempTankSensorError	:= StatusTemperatureInput(X20AT4222_216.Status01, 1);
	gInksInputs[9].iTemperatureTankRaw			:= X20AT4222_216.TempInput[2];
	gInksInputs[9].xTempTankSensorError	:= StatusTemperatureInput(X20AT4222_216.Status01, 2);
	gInksInputs[8].iTemperatureTankRaw			:= X20AT4222_216.TempInput[3];
	gInksInputs[8].xTempTankSensorError	:= StatusTemperatureInput(X20AT4222_216.Status01, 3);
	gInksInputs[7].iTemperatureTankRaw			:= X20AT4222_216.TempInput[4];
	gInksInputs[7].xTempTankSensorError	:= StatusTemperatureInput(X20AT4222_216.Status01, 4);

	// X20SI8110_217
	gBlockInputs[2].Safety.xRearEStopOK:=X20SI8110_217.DInput[1];
	gBlockInputs[2].Safety.xFrontEStopOK:=X20SI8110_217.DInput[3];
	gBlockInputs[2].Safety.xCurtainEnable01:=X20SI8110_217.DInput[5];
	gBlockInputs[2].Safety.xRearSafetyOK:=X20SI8110_217.DInput[6];
	gBlockInputs[2].Safety.xCurtainEnable02:=X20SI8110_217.DInput[7];

	gBlockInputs[2].Safety.xSafetyOK:=X20SO2110_218.DInput[1];

	// SI UNIT BK2
	gBlockInputs[2].xSiUnitModuleOk:= SiUnitBK2.ModuleOk;  // Filter if it's necesary
	////Reserve01.DInput[1]:= SiUnitBK2.Input01_08.0;
	gBlockInputs[2].xAirVenturiOK:= SiUnitBK2.Input01_08.1;
	gBlockInputs[2].xTrayOut:=  SiUnitBK2.Input01_08.2;   //Out: Tray in safe position to move bars to print
	gBlockInputs[2].xIclaSensor:= SiUnitBK2.Input01_08.3;

	//Signals Forced by Configuration

	gMachine.In.x24Vdc				:= TRUE;

	FOR iIndexBlock := 1 TO gMachine.Pt.CT.iNumBlocks DO

		gBlockInputs[iIndexBlock].Safety.xFrontSafetyOK	:= TRUE;

		gBlockInputs[iIndexBlock].xHeaterDcOkBusBar2 := TRUE;
		gBlockInputs[iIndexBlock].xModuleTemp04Ok := TRUE;

		gBlock[iIndexBlock].parameters.Hw.iNumPrintheadsPSU := 0;
		gBlock[iIndexBlock].parameters.Hw.iNumHeaterPSU := 0;

	END_FOR

END_ACTION
```

#### InputsShield.st
```iecst
ACTION InputsShield:

(* CABINET 01 *)

	//X1 PLC

	// Those variables are not mapped. Are fast and assigned with pointer
	//	gPhotoCells.Inputs.Signals.xPhotoCells[1]	:= NOT X1.DInput[1];
	//	gPhotoCells.Inputs.Signals.xPhotoCells[2]	:= NOT X1.DInput[2];
	//	gPhotoCells.Inputs.Signals.xPhotoCells[3]	:= NOT X1.DInput[3];

	gBlockInputs[1].xReferenceDI			:= X1.DInput[4];

	//X2 PLC
	gBelt.parameters.xDriveProtectionOK			:= X2.DInput[1];
	gBlockInputs[1].xDriveProtectionOK			:= X2.DInput[2];
	gBlockInputs[1].xDifferentialOK				:= X2.DInput[3];
	gMachine.In.xCoolingPCSensorAlrm			:= X2.DInput[4];
	gMachine.In.ProductDetect.pPDSignalSensorL1	:= ADR(X2.DInput[5]);
	gMachine.In.ProductDetect.pPDSignalSensorL2	:= ADR(X2.DInput[6]);
	gMachine.In.UPSs[1].xSystemFault			:= NOT X2.DInput[7];
	gMachine.In.UPSs[1].xPowerFault				:= NOT X2.DInput[8];
	gMachine.In.UPSs[1].xLowBattery					:= NOT X2.DInput[9];
	gMachine.In.UPSs[1].xByPass					:= NOT X2.DInput[10];

	// X20DIF371_001
	gInksInputs[1].xKlixonTriggered		:= X20DIF371_001.DInput[1];
	gInksInputs[2].xKlixonTriggered		:= X20DIF371_001.DInput[2];
	gInksInputs[1].xMinLevel			:= X20DIF371_001.DInput[3];
	gInksInputs[2].xMinLevel			:= X20DIF371_001.DInput[4];
	gInksInputs[1].xMaxLevel			:= X20DIF371_001.DInput[5];
	gInksInputs[2].xMaxLevel			:= X20DIF371_001.DInput[6];
	gInksInputs[1].xOverpressure 		:= NOT X20DIF371_001.DInput[7];
	gInksInputs[2].xOverpressure 		:= NOT X20DIF371_001.DInput[8];
	//Reserve01.DInput[1]					:= X20DIF371_001.DInput[9];
	//Reserve01.DInput[1]					:= X20DIF371_001.DInput[10];
	//Reserve01.DInput[1]					:= X20DIF371_001.DInput[11];
	//Reserve01.DInput[1]					:= X20DIF371_001.DInput[12];
	//Reserve01.DInput[1]					:= X20DIF371_001.DInput[13];
	gBlockInputs[1].xHeaterDcOkBusBar1	:= X20DIF371_001.DInput[14];
	gInksInputs[1].xPrintHeadsPsuOK		:= X20DIF371_001.DInput[15];
	gInksInputs[2].xPrintHeadsPsuOK		:= X20DIF371_001.DInput[16];

	// X20DIF371_002
	gMachine.In.xConsentL1Ok			:= X20DIF371_002.DInput[1];
	gMachine.In.xConsentL2Ok			:= X20DIF371_002.DInput[2];
	gMachine.In.xExternalCleaningOrder	:= X20DIF371_002.DInput[3];
	//Reserve01.DInput[1]					:= X20DIF371_002.DInput[4];
	gMachine.In.Buttons.xStart					:= X20DIF371_002.DInput[5];
	gMachine.In.Buttons.xStop					:= NOT X20DIF371_002.DInput[6];
	gMachine.In.Buttons.xAuto					:= X20DIF371_002.DInput[7];
	gMachine.In.Buttons.xZero					:= NOT X20DIF371_002.DInput[8];
	gMachine.In.Buttons.xManual					:= X20DIF371_002.DInput[9];
	//gMachine.In.Buttons.xReset					:= X20DIF371_002.DInput[10];

	// gMachine.In.iMachineModelCode assigned in an specific Action

	//Reserve01.DInput[1] 				:= X20DIF371_002.DInput[15];
	//Reserve01.DInput[1] 				:= X20DIF371_002.DInput[16];

	// Reset and Mute with the same digital signal
	T_Reset.IN := X20DIF371_002.DInput[10];
	T_Reset.PT := t#250ms;
	T_Reset();

	T_Mute.IN := X20DIF371_002.DInput[10];
	T_Mute.PT := t#100ms;
	T_Mute();

	gMachine.In.Buttons.xReset:= T_Reset.Q;
	gMachine.In.Buttons.xMute:= T_Mute.Q;

	// X20DIF371_003
	gMachine.In.ProductDetect.pPDCarriageSignalL1 := ADR(X20DIF371_003.DInput[1]);
	gMachine.In.ProductDetect.pPDCarriageSignalL2 := ADR(X20DIF371_003.DInput[2]);
	Reserve01.DInput[3] 				:= X20DIF371_003.DInput[3];
	gMachine.In.xPC2Ok 					:= X20DIF371_003.DInput[4];
	//Reserve01.DInput[1] 				:= X20DIF371_003.DInput[5];
	//Reserve01.DInput[1] 				:= X20DIF371_003.DInput[6];
	//Reserve01.DInput[1]					:= X20DIF371_003.DInput[7];
	gMachine.In.xPbfCardOK 				:= X20DIF371_003.ModuleOk;
	gMachine.In.iRelieve1.0 			:= X20DIF371_003.DInput[8];
	gMachine.In.iRelieve1.1 			:= X20DIF371_003.DInput[9];
	gMachine.In.iRelieve1.2 			:= X20DIF371_003.DInput[10];
	gMachine.In.iRelieve1.3 			:= X20DIF371_003.DInput[11];
	gMachine.In.iRelieve1.4 			:= X20DIF371_003.DInput[12];
	gMachine.In.iRelieve1.5 			:= X20DIF371_003.DInput[13];
	gMachine.In.iRelieve1.6 			:= X20DIF371_003.DInput[14];
	gMachine.In.iRelieve1.7 			:= X20DIF371_003.DInput[15];
	gMachine.In.iRelieve1.8 			:= X20DIF371_003.DInput[16];

	// X20DIF371_004
	gChiller[1].In.xPowered				:= X20DIF371_004.DInput[1];
	gChiller[1].In.xCooling 			:= X20DIF371_004.DInput[1]; //xCooling input was asked in Nz2AQ but Shield's chiller has no cooling output. So assuming "Powered"="Running"
	gChiller[1].In.xAlarm	 			:= NOT X20DIF371_004.DInput[2];
	gBlockInputs[1].xWaterLevelSensor 	:= X20DIF371_004.DInput[3];
	gBlockInputs[1].xWaterPresureSensor	:= X20DIF371_004.DInput[4];
	//Reserve01.DInput[1] 				:= X20DIF371_004.DInput[5];
	//Reserve01.DInput[1] 				:= X20DIF371_004.DInput[6];
	//Reserve01.DInput[1] 				:= X20DIF371_004.DInput[7];
	//Reserve01.DInput[1] 				:= X20DIF371_004.DInput[8];
	gBlockInputs[1].Safety.xSafetyOK	  		:= X20DIF371_004.DInput[9];
	gBlockInputs[1].Safety.xFrontSafetyOK 		:= X20DIF371_004.DInput[10];
	gBlockInputs[1].Safety.xRearSafetyOK 		:= X20DIF371_004.DInput[11];
	//Reserve01.DInput[1] 				:= X20DIF371_004.DInput[12];
	//Reserve01.DInput[1] 				:= X20DIF371_004.DInput[13];
	//Reserve01.DInput[1] 				:= X20DIF371_004.DInput[14];
	//Reserve01.DInput[1] 				:= X20DIF371_004.DInput[15];
	//Reserve01.DInput[1] 				:= X20DIF371_004.DInput[16];

	// X20AI4322_008	(* BAR A *)		(* BAR B *)
	gInksInputs[1].iVacuum1Raw			:= X20AI4322_008.AInput[1];
	gInksInputs[1].xVacuum1SensorError	:= StatusAnalogInputBroken( X20AI4322_008.ModuleOk, X20AI4322_008.Status01, 0, 1);
	gInksInputs[2].iVacuum1Raw			:= X20AI4322_008.AInput[2];
	gInksInputs[2].xVacuum1SensorError	:= StatusAnalogInputBroken( X20AI4322_008.ModuleOk, X20AI4322_008.Status01, 0, 2);
	gInksInputs[1].iVacuum2Raw			:= X20AI4322_008.AInput[3];
	gInksInputs[1].xVacuum2SensorError	:= StatusAnalogInputBroken( X20AI4322_008.ModuleOk, X20AI4322_008.Status01, 0, 3);
	gInksInputs[2].iVacuum2Raw			:= X20AI4322_008.AInput[4];
	gInksInputs[2].xVacuum2SensorError	:= StatusAnalogInputBroken( X20AI4322_008.ModuleOk, X20AI4322_008.Status01, 0, 4);

	// X20AT4222_010
	gBlockInputs[1].xModuleTemp01Ok		:= X20AT4222_010.ModuleOk;
	gInksInputs[1].iTemperatureRaw		:= X20AT4222_010.TempInput[1];
	gInksInputs[1].xTempSensorError		:= StatusTemperatureInput(X20AT4222_010.Status01, 1);
	gInksInputs[2].iTemperatureRaw		:= X20AT4222_010.TempInput[2];
	gInksInputs[2].xTempSensorError		:= StatusTemperatureInput(X20AT4222_010.Status01, 2);
	gChiller[1].In.WaterManifold.iEnvironmentTempRaw	:= X20AT4222_010.TempInput[3];
	gChiller[1].In.WaterManifold.xTempEnvSensError	:= StatusTemperatureInput(X20AT4222_010.Status01, 3);
	gChiller[1].In.WaterManifold.iWaterManifoldTempRaw	:= X20AT4222_010.TempInput[4];
	gChiller[1].In.WaterManifold.xTempWatSensError	:= StatusTemperatureInput(X20AT4222_010.Status01, 4);

	// X20SM1436_11
	gPhotoCells.status.xBackModuleOk := X20SM1436_011.ModuleOk;

	// X20SM1436_12
	gPhotoCells.status.xFrontModuleOk := X20SM1436_012.ModuleOk;

	// SI UNIT BK1
	gBlockInputs[1].xSiUnitModuleOk		:= SiUnitBK1.ModuleOk;  // Filter if it's necesary
	gMachine.In.xAirSupply				:= SiUnitBK1.Input01_08.0;
	gBlockInputs[1].xAirVenturiOK		:= SiUnitBK1.Input01_08.1;
	gBlockInputs[1].xTrayOut			:= SiUnitBK1.Input01_08.2;
	gBlockInputs[1].xIclaSensor			:= SiUnitBK1.Input01_08.3;
	gBlockInputs[1].xBarsIn := TRUE;

	//Signals Forced by Configuration
	gMachine.In.UPSs[2].xPowerFault		:= FALSE;
	gMachine.In.UPSs[2].xByPass			:= FALSE;
	gMachine.In.UPSs[2].xLowBattery			:= FALSE;
	gMachine.In.UPSs[2].xSystemFault	:= FALSE;
	gMachine.In.xPC1Ok				:= TRUE;
	gMachine.In.x24Vdc				:= TRUE;

	FOR iIndexBlock := 1 TO gMachine.Pt.CT.iNumBlocks DO

		gBlockInputs[iIndexBlock].Safety.xCurtainEnable01:= TRUE;
		gBlockInputs[iIndexBlock].Safety.xCurtainEnable02:= TRUE;
		gBlockInputs[iIndexBlock].Safety.xFrontEStopOK := TRUE;
		gBlockInputs[iIndexBlock].Safety.xRearEStopOK	:= TRUE;

		gBlockInputs[iIndexBlock].xModuleTemp02Ok	:= TRUE;
		gBlockInputs[iIndexBlock].xModuleTemp03Ok := TRUE;
		gBlockInputs[iIndexBlock].xModuleTemp04Ok := TRUE;

		gBlockInputs[iIndexBlock].xHeaterDcOkBusBar2 := TRUE;

		gBlock[iIndexBlock].parameters.Hw.iNumPrintheadsPSU := 0;
		gBlock[iIndexBlock].parameters.Hw.iNumHeaterPSU := 0;

	END_FOR

END_ACTION
```

#### MappingInputs.st
```iecst
PROGRAM _CYCLIC

	//If in automation runtime, do not assign physical mapping
	IF gMachine.St.HwData.Family = FAMILY_BRAUTOMATIONRUNTIME THEN
		RETURN;
	END_IF

	CASE gMachine.Pt.MachineModel OF
		Type_P4_6B,
		Type_P4_6B_L,
		Type_P4_12B,
		Type_P4_12B_L:
			InputsP4;

		Type_SHLD,
		Type_SHLD_L:
			InputsShield;

		Type_S1400,
		Type_S1400_VAC_PWRLNK,
		Type_S1400_VAC_CAN:
			InputsS1400;

		Type_P5_OIL,
		Type_P5_WTR:
			InputsP5;

		Type_NOZ_2_AQ,
		Type_NOZ_2_UV,
		Type_NOZ_2_UV_White:
			InputsNozomi2;

		Type_CUBE,
		Type_CUBE_INSPECTION,
		Type_CUBE_GULLIVER,
		Type_CUBE_GULLIVER_INSPECTION:
			InputsCube;

		Type_MECANO_UV_WHITE,
		Type_MECANO_UV_OPV,
		Type_MECANO_UV_WHITE_OPV:
			InputsMecano;

	END_CASE

END_PROGRAM
```

### Program Logical/Printer/PhysicalMapping/PhysicalMapOutputs (IEC) - Physical outputs assignation

#### OutputsNozomi2.st
```iecst
ACTION OutputsNozomi2:

	//////////
	//PRINTER
	//////////
	X20DOF322_108.DOutput[1] := gBlockOutputs[1].xShotLine1;
	X20DOF322_108.DOutput[2] := gBlockOutputs[1].xShotLine2;
	X20DOF322_108.DOutput[3] := gBlockOutputs[1].xEnableDobleShot;
	X20DOF322_108.DOutput[4] := gMachine.Out.xResetCB1;
	X20DOF322_108.DOutput[5] := gMachine.Out.xResetRouter;
	X20DOF322_108.DOutput[6] := gThicknessCtrl.Outputs.xEnableMediaSignalToCb;
	X20DOF322_108.DOutput[7] := gMachine.Out.xAirSupply;
	X20DOF322_108.DOutput[8] := gLine.Outputs.xGreenLight;
	X20DOF322_108.DOutput[9] := gLine.Outputs.xLightReset OR gMachine.Out.xLightReset;;
	X20DOF322_108.DOutput[10] := gLine.Outputs.xSound OR gMachine.Out.xBuzzerButtonPanel;
	X20DOF322_108.DOutput[11] := gLine.Outputs.xSound OR gMachine.Out.xBuzzerButtonPanel;
	X20DOF322_108.DOutput[12] := gLine.Outputs.xYellowLight;
	X20DOF322_108.DOutput[13] := gLine.Outputs.xBlueLight;
	X20DOF322_108.DOutput[14] := gLine.Outputs.xRedLight;
	X20DOF322_108.DOutput[15] := gLine.Outputs.xWhiteLight;

	X20DOF322_109.DOutput[1] := gInksOutputs[1].xOutPowPrintHead;
	X20DOF322_109.DOutput[2] := gInksOutputs[2].xOutPowPrintHead;
	X20DOF322_109.DOutput[3] := gInksOutputs[3].xOutPowPrintHead;
	X20DOF322_109.DOutput[4] := gInksOutputs[4].xOutPowPrintHead;
	X20DOF322_109.DOutput[5] := gInksOutputs[5].xOutPowPrintHead;
	X20DOF322_109.DOutput[6] := gInksOutputs[6].xOutPowPrintHead;
	X20DOF322_109.DOutput[7] := gInksOutputs[7].xOutPowPrintHead;
	X20DOF322_109.DOutput[8] := gInksOutputs[8].xOutPowPrintHead;
	X20DOF322_109.DOutput[9] := gInksOutputs[1].xOutBarResistance;
	X20DOF322_109.DOutput[10] := gInksOutputs[2].xOutBarResistance;
	X20DOF322_109.DOutput[11] := gInksOutputs[3].xOutBarResistance;
	X20DOF322_109.DOutput[12] := gInksOutputs[4].xOutBarResistance;
	X20DOF322_109.DOutput[13] := gInksOutputs[5].xOutBarResistance;
	X20DOF322_109.DOutput[14] := gInksOutputs[6].xOutBarResistance;
	X20DOF322_109.DOutput[15] := gInksOutputs[7].xOutBarResistance;
	X20DOF322_109.DOutput[16] := gInksOutputs[8].xOutBarResistance;

	X20DOF322_110.DOutput[1] := gJamDetect[1].Outputs.xJamTestSignal[1] OR
								gJamDetect[2].Outputs.xJamTestSignal[1] OR
								gJamDetect[3].Outputs.xJamTestSignal[1];
	X20DOF322_110.DOutput[2] := gJamDetect[1].Outputs.xJamTestSignal[2] OR
								gJamDetect[2].Outputs.xJamTestSignal[2] OR
								gJamDetect[3].Outputs.xJamTestSignal[2];
	X20DOF322_110.DOutput[3] := gJamDetect[1].Outputs.xJamTestSignal[3] OR
								gJamDetect[2].Outputs.xJamTestSignal[3] OR
								gJamDetect[3].Outputs.xJamTestSignal[3];
	X20DOF322_110.DOutput[4] := gJamDetect[1].Outputs.xJamTestSignal[4] OR
								gJamDetect[2].Outputs.xJamTestSignal[4] OR
								gJamDetect[3].Outputs.xJamTestSignal[4];
	X20DOF322_110.DOutput[5] := gMachine.Out.xRemoteTeachL1;
	X20DOF322_110.DOutput[6] := gMachine.Out.xRemoteTeachL2;
	X20DOF322_110.DOutput[7] := gMachine.Out.xDegasser;

	// NOZOMITWO-2541 For advance team testing on Alpha
	IF (gMachine.Pt.MachineModel = Type_NOZ_2_AQ) THEN
		X20DOF322_110.DOutput[9] := gInks[2].signals.out.xSolenoid1;
		X20DOF322_110.DOutput[10] := gInks[2].signals.out.xSolenoid2;
		X20DOF322_110.DOutput[11] := gInks[2].signals.out.xSolenoid3;
		X20DOF322_110.DOutput[12] := gInks[2].signals.out.xSolenoid4;
	END_IF

	//Analog outputs
	X20AO4622_115.AOutput[1] := gInksOutputs[2].iDutyCycleNegative;
	X20AO4622_115.AOutput[2] := gInksOutputs[3].iDutyCycleNegative;
 	X20AO4622_115.AOutput[3] := gInksOutputs[2].iDutyCycleFilling;
	X20AO4622_115.AOutput[4] := gInksOutputs[3].iDutyCycleFilling;
 	X20AO4622_116.AOutput[1] := gInksOutputs[4].iDutyCycleNegative;
	X20AO4622_116.AOutput[2] := gInksOutputs[5].iDutyCycleNegative;
 	X20AO4622_116.AOutput[3] := gInksOutputs[4].iDutyCycleFilling;
	X20AO4622_116.AOutput[4] := gInksOutputs[5].iDutyCycleFilling;
	X20AO4622_117.AOutput[1] := gInksOutputs[6].iDutyCycleNegative;

	IF (gMachine.Pt.MachineModel = Type_NOZ_2_AQ) THEN
		X20AO4622_117.AOutput[2] := gInksOutputs[7].iDutyCycleNegative;
	ELSE
		X20AO4622_117.AOutput[2] := gInksOutputs[8].iDutyCycleNegative;
	END_IF

	X20AO4622_117.AOutput[3] := gInksOutputs[6].iDutyCycleFilling;

	IF (gMachine.Pt.MachineModel = Type_NOZ_2_AQ) THEN
		X20AO4622_117.AOutput[4] := gInksOutputs[7].iDutyCycleFilling;
	ELSE
		X20AO4622_117.AOutput[4] := gInksOutputs[8].iDutyCycleFilling;
	END_IF

	///////////////////////////
	//UV Curing leds related

	//Digital outputs
	X20DOF322_155.DOutput[1] := gMachine.commands.CleanBelt.xCleanBeltMoveFwd;
	X20DOF322_155.DOutput[2] := gMachine.commands.CleanBelt.xCleanBeltMoveBwd;
	X20DOF322_155.DOutput[3] := gMachine.commands.CleanBelt.xCleanBeltResetRelay;
	X20DOF322_155.DOutput[5] := gCuringLed[iIndexColorCuringLedBar].Lamp[1].Outputs.EnableLamp;
	X20DOF322_155.DOutput[6] := gCuringLed[iIndexColorCuringLedBar].Lamp[2].Outputs.EnableLamp;
	X20DOF322_155.DOutput[7] := gCuringLed[iIndexColorCuringLedBar].Lamp[3].Outputs.EnableLamp;
	X20DOF322_155.DOutput[8] := gCuringLed[iIndexColorCuringLedBar].Lamp[4].Outputs.EnableLamp;
	X20DOF322_155.DOutput[9] := gCuringLed[iIndexWhiteCuringLedBar].Lamp[1].Outputs.EnableLamp;
	X20DOF322_155.DOutput[10] := gCuringLed[iIndexWhiteCuringLedBar].Lamp[2].Outputs.EnableLamp;
	X20DOF322_155.DOutput[11] := gCuringLed[iIndexWhiteCuringLedBar].Lamp[3].Outputs.EnableLamp;
	X20DOF322_155.DOutput[12] := gCuringLed[iIndexWhiteCuringLedBar].Lamp[4].Outputs.EnableLamp;
	X20DOF322_155.DOutput[15] := gMachine.Out.xAntiStaticPOn;

	//Analog outputs
	X20AO4622_157.AOutput[1] := gCuringLed[iIndexColorCuringLedBar].Lamp[1].Outputs.IntensityLampRaw;
	X20AO4622_157.AOutput[2] := gCuringLed[iIndexColorCuringLedBar].Lamp[2].Outputs.IntensityLampRaw;
	X20AO4622_157.AOutput[3] := gCuringLed[iIndexColorCuringLedBar].Lamp[3].Outputs.IntensityLampRaw;
	X20AO4622_157.AOutput[4] := gCuringLed[iIndexColorCuringLedBar].Lamp[4].Outputs.IntensityLampRaw;

	X20AO4622_158.AOutput[1] := gCuringLed[iIndexWhiteCuringLedBar].Lamp[1].Outputs.IntensityLampRaw;
	X20AO4622_158.AOutput[2] := gCuringLed[iIndexWhiteCuringLedBar].Lamp[2].Outputs.IntensityLampRaw;
	X20AO4622_158.AOutput[3] := gCuringLed[iIndexWhiteCuringLedBar].Lamp[3].Outputs.IntensityLampRaw;
	X20AO4622_158.AOutput[4] := gCuringLed[iIndexWhiteCuringLedBar].Lamp[4].Outputs.IntensityLampRaw;

	//////////
	//PDC
	//////////
	//Pdc_X20DOF322_008.DOutput
	Pdc_X20DOF322_008.DOutput[1] := gLine.Outputs.ExternalDevices[2].xClose;
	Pdc_X20DOF322_008.DOutput[2] := gLine.Outputs.ExternalDevices[1].xClose;
	Pdc_X20DOF322_008.DOutput[3] := gLine.Outputs.ExternalDevices[1].xOpen;
	Pdc_X20DOF322_008.DOutput[4] := gLine.Outputs.ExternalDevices[10].xClose;
	Pdc_X20DOF322_008.DOutput[5] := gLine.Outputs.ExternalDevices[10].xOpen;
	Pdc_X20DOF322_008.DOutput[6] := gLine.Outputs.ExternalDevices[0].xClose AND gMachine.In.xPowerSwitch;
	Pdc_X20DOF322_008.DOutput[7] := gLine.Outputs.ExternalDevices[6].xClose;
	Pdc_X20DOF322_008.DOutput[8] := gMachine.Out.xSuctionTurbine; //gLine.Outputs.ExternalDevices[9].xClose;
	Pdc_X20DOF322_008.DOutput[9] := gLine.Outputs.ExternalDevices[8].xClose;
	Pdc_X20DOF322_008.DOutput[10] := gLine.Outputs.ExternalDevices[7].xClose;
	Pdc_X20DOF322_008.DOutput[11] := gLine.Outputs.ExternalDevices[3].xClose;
	Pdc_X20DOF322_008.DOutput[12] := gLine.Outputs.ExternalDevices[3].xOpen;
	Pdc_X20DOF322_008.DOutput[13] := gLine.Outputs.ExternalDevices[4].xClose;
	Pdc_X20DOF322_008.DOutput[14] := gLine.Outputs.ExternalDevices[4].xOpen;
	Pdc_X20DOF322_008.DOutput[15] := gLine.Outputs.ExternalDevices[5].xClose;
	Pdc_X20DOF322_008.DOutput[16] := gMachine.Out.xResetRouter;

	//Pdc_X20DOF322_009
	//Pdc_X20DOF322_009.DOutput[1] := Reset Hub Powerlink PDC;
	Pdc_X20DOF322_009.DOutput[2] := gMachine.St.Remote.xSafetyReadyToReset;
	Pdc_X20DOF322_009.DOutput[3] := gLine.Outputs.Customer[1];
	Pdc_X20DOF322_009.DOutput[4] := gLine.Outputs.Customer[2];
	Pdc_X20DOF322_009.DOutput[5] := gLine.Outputs.Customer[3];
	Pdc_X20DOF322_009.DOutput[6] := gFeeder.Outputs.Physical.xPrepareToFeed;
	Pdc_X20DOF322_009.DOutput[7] := gFeeder.Outputs.Physical.xStartFeeding;
	Pdc_X20DOF322_009.DOutput[8] := gFeeder.Outputs.Physical.xFastStop;
	Pdc_X20DOF322_009.DOutput[9] := gPrimer.Outputs.Physical.xRunDryer;
	Pdc_X20DOF322_009.DOutput[10] := gPrimer.Outputs.Physical.xRunTransport;
	Pdc_X20DOF322_009.DOutput[11] := gPrimer.Outputs.Physical.xRunPriming;
	Pdc_X20DOF322_009.DOutput[12] := gPrimer.Outputs.Physical.xPrepareToPrime;
	Pdc_X20DOF322_009.DOutput[13] := gStacker.Outputs.xRun;
	Pdc_X20DOF322_009.DOutput[14] := gThicknessCtrl.Outputs.xReject;
	Pdc_X20DOF322_009.DOutput[15] := gStacker.Outputs.xPrepareToStack;
	Pdc_X20DOF322_009.DOutput[16] := gStacker.Outputs.xEjectRejectStack;

	//Pdc_X20DOF322_010
	Pdc_X20DOF322_010.DOutput[1] := gStacker.Outputs.xStackEject;
	Pdc_X20DOF322_010.DOutput[2] := gLine.Outputs.ExternalDevices[5].xClose; //To review how UPS for dryer should be activated
	Pdc_X20DOF322_010.DOutput[3] := gOverVarnish.Outputs.Physical.xRunDryer;
	Pdc_X20DOF322_010.DOutput[4] := gOverVarnish.Outputs.Physical.xRunTransport;
	Pdc_X20DOF322_010.DOutput[5] := gOverVarnish.Outputs.Physical.xRunPriming;
	Pdc_X20DOF322_010.DOutput[6] := gOverVarnish.Outputs.Physical.xPrepareToPrime;
	Pdc_X20DOF322_010.DOutput[7] := gLine.Outputs.ExternalDevices[0].xClose AND gMachine.In.xPowerSwitch;
	Pdc_X20DOF322_010.DOutput[8] := gLine.Outputs.ExternalDevices[0].xClose;
	Pdc_X20DOF322_010.DOutput[9] := gLine.Outputs.ExternalDevices[0].xClose;
	Pdc_X20DOF322_010.DOutput[10] := gBeltClean.Outputs.xAirTurbineOn; // NOZOMITWO-1912
	Pdc_X20DOF322_010.DOutput[11] := gBeltClean.Outputs.xAirTurbineVSDReset; // NOZOMITWO-1912
	Pdc_X20DOF322_010.DOutput[12] := gDryerAnc.Outputs.xRunTransport;
	(*
	Pdc_X20DOF322_010.DOutput[13] := ;
	Pdc_X20DOF322_010.DOutput[14] := ;
	Pdc_X20DOF322_010.DOutput[15] := ;
	*)
	Pdc_X20DOF322_010.DOutput[16] := gChiller[1].Out.xStart; // NOZOMITWO-2428 Only for Noz2 water, normally the start signal is a feedback of the Chiller PowerOn CB or is not needed

	//Line X20DOF322_023
	Pdc_X20DOF322_023.DOutput[1] := gChiller[gCuringLed[iIndexColorCuringLedBar].Parameters.iChillerIndex].Out.xStart; //gCuringLed[iIndexColorCuringLedBar].Signals.Outputs.xRunChiller;
	Pdc_X20DOF322_023.DOutput[2] := gChiller[gCuringLed[iIndexWhiteCuringLedBar].Parameters.iChillerIndex].Out.xStart; //gCuringLed[iIndexWhiteCuringLedBar].Signals.Outputs.xRunChiller;
	Pdc_X20DOF322_023.DOutput[3] := gLine.Outputs.ExternalDevices[7].xClose AND gCuringLed[iIndexColorCuringLedBar].Signals.Outputs.xPowerOnLamps AND NOT gSafetyController.Alarms.xAlrPrinter AND gLine.Inputs.xPrinterPowered; //UV leds color power
	Pdc_X20DOF322_023.DOutput[4] := gLine.Outputs.ExternalDevices[7].xClose AND gCuringLed[iIndexWhiteCuringLedBar].Signals.Outputs.xPowerOnLamps AND NOT gSafetyController.Alarms.xAlrPrinter AND gLine.Inputs.xPrinterPowered; //UV leds white power
	Pdc_X20DOF322_023.DOutput[5] := gLine.Outputs.ExternalDevices[8].xClose AND NOT gSafetyController.Alarms.xAlrPrinter; //Chiller color power
	Pdc_X20DOF322_023.DOutput[6] := gLine.Outputs.ExternalDevices[8].xClose AND NOT gSafetyController.Alarms.xAlrPrinter; //Chiller white power

	//Line X20DOF322_051
	//Pdc_X20DOF322_051.DOutput[1] := ;
	Pdc_X20DOF322_051.DOutput[1] := gSarm.Outputs.xStartTransport;
	Pdc_X20DOF322_051.DOutput[2] := gSarm.Outputs.xFastStop;
	Pdc_X20DOF322_051.DOutput[4] := gLine.Outputs.ExternalDevices[11].xClose; // DG SARM
	Pdc_X20DOF322_051.DOutput[5] := gLine.Outputs.ExternalDevices[1].xClose; // DG InfraRed Primer TecLighting

	// SI UNIT BK1
	SiUnitPwrLnkBK1.Output01_16.0 := 	gBlockOutputs[1].xTrayIn; //1A
	SiUnitPwrLnkBK1.Output01_16.1 := 	gBlockOutputs[1].xTrayOut; //1B
	SiUnitPwrLnkBK1.Output01_16.2 := 	gMachine.commands.CleanBelt.xCleanBeltPump OR
										gCuringLed[1].Signals.Outputs.xPowerOnNitrogen OR
										gCuringLed[2].Signals.Outputs.xPowerOnNitrogen OR
										gBeltClean.Outputs.xPumpOn;  //2A //[RGP] This EV has different purposes in UV and Water // NOZOMITWO-1912
	SiUnitPwrLnkBK1.Output01_16.3 := 	gBlockOutputs[1].xVenturi; //2B
	//SiUnitPwrLnkBK1.Output01_16.4 :=  //3A
	SiUnitPwrLnkBK1.Output01_16.5 := 	gMachine.commands.CleanBelt.xPistonFlojet OR gBeltClean.Outputs.xRiseCleaningSystem;  //4A // NOZOMITWO-1912
	SiUnitPwrLnkBK1.Output01_16.6 := 	FALSE; //5A
	SiUnitPwrLnkBK1.Output01_16.7 := 	gBlockOutputs[1].xWastedInkTankPump; //6A

	//Vacuum
	SiUnitPwrLnkBK1.Output01_16.8 := gTransVacuum[1].Outputs.VacuumValves.0;	//10A
	SiUnitPwrLnkBK1.Output01_16.9 := gTransVacuum[1].Outputs.VacuumValves.1;	//10B
	SiUnitPwrLnkBK1.Output01_16.10 := gTransVacuum[1].Outputs.VacuumValves.2;	//11A
	SiUnitPwrLnkBK1.Output01_16.11 := gTransVacuum[1].Outputs.VacuumValves.3;	//11B
	SiUnitPwrLnkBK1.Output01_16.12 := gTransVacuum[1].Outputs.VacuumValves.4;	//12A
	SiUnitPwrLnkBK1.Output01_16.13 := gTransVacuum[1].Outputs.VacuumValves.5;	//12B
	SiUnitPwrLnkBK1.Output01_16.14 := gTransVacuum[1].Outputs.VacuumValves.6;	//13A
	SiUnitPwrLnkBK1.Output01_16.15 := gTransVacuum[1].Outputs.VacuumValves.7;	//13B
	SiUnitPwrLnkBK1.Output17_32.0 := gTransVacuum[1].Outputs.VacuumValves.8;	//14A
	SiUnitPwrLnkBK1.Output17_32.1 := gTransVacuum[1].Outputs.VacuumValves.9;	//14B
	SiUnitPwrLnkBK1.Output17_32.2 := gTransVacuum[1].Outputs.VacuumValves.10;	//15A
	SiUnitPwrLnkBK1.Output17_32.3 := gTransVacuum[1].Outputs.VacuumValves.11;	//15B
	SiUnitPwrLnkBK1.Output17_32.4 := gTransVacuum[1].Outputs.VacuumValves.12;	//16A
	SiUnitPwrLnkBK1.Output17_32.5 := gTransVacuum[1].Outputs.VacuumValves.13;	//16B
	SiUnitPwrLnkBK1.Output17_32.6 := gTransVacuum[1].Outputs.VacuumValves.14;	//17A From 17A to 19B: removed, but not in old machines.
	SiUnitPwrLnkBK1.Output17_32.7 := gTransVacuum[1].Outputs.VacuumValves.15;	//17B
	SiUnitPwrLnkBK1.Output17_32.8 := gTransVacuum[1].Outputs.VacuumValves.16;	//18A
	SiUnitPwrLnkBK1.Output17_32.9 := gTransVacuum[1].Outputs.VacuumValves.17;	//18B
	SiUnitPwrLnkBK1.Output17_32.10 := gTransVacuum[1].Outputs.VacuumValves.18;	//19A
	SiUnitPwrLnkBK1.Output17_32.11 := gTransVacuum[1].Outputs.VacuumValves.19;	//19B

END_ACTION
```
